FUNCTION_BLOCK "RECEIVER"	// FB 1011
TITLE = REC01
//Creation:
//Date:            Author:                                               Version
//--------------------------------------------------------------------------------
//14.04.2018     Ilia Bedniakov (ilia)                                   01.00.00
//
//Changes:
//No. Date:        Who       Description                           Mark   Version 
//--------------------------------------------------------------------------------
//01  12.01.2019  ilia       correction at comissioning            (001)  01.01.00
//
//
//_______________________________________________________________________________
//Function:
AUTHOR : ilia
NAME : project
VERSION : 0.1
VAR_INPUT
  I_iIFVacuumPumpDB : INT ;	//VacuumPump DB Nr
  I_iIFVacuumPumpDW : INT ;	//VacuumPump Interface Start DW Nr
  I_iIFStorageDB : INT ;
  I_iIFStorageDW : INT ;
  I_iIFStoLocParDB : INT ;
  I_xSystemActive : BOOL ;	//system control on
  I_xAngleValveOpen : BOOL ;	//Angle Valve Close
  I_xAngleValveClose : BOOL ;	//Angle Valve Close
  i_xPendelFlapREC : BOOL ;	//Pendulum Flap
  i_xHighLevelREC : BOOL ;	//high level sensor
  I_xPFC_PM1 : BOOL ;	//PFC PM Hopper Big Components
  I_xPFC_PM2 : BOOL ;	//PFC PM Hopper Small Components
  i_xAckFullReceiver : BOOL ;
  i_xAngleValve : BOOL ;
END_VAR
VAR_IN_OUT
  q_xAngleValve : BOOL ;	//Angle Valve Open
  q_xCleaningValve : BOOL ;	//Filter Cleaning Valve
  q_xRepperValve : BOOL ;	//Rapper Valve
  q_xRedLamp : BOOL ;
  q_xYellowLamp : BOOL ;
  q_xGreenLamp : BOOL ;
  f_xAngleValve : BOOL ;	//Angle Valve Open
  f_xFullReceiver : BOOL ;	//Fault
  f_xNoStartConditions : BOOL ;
  f_xNoPFCRequest : BOOL ;
END_VAR
VAR
  reserve_IO : ARRAY  [14 .. 49 ] OF BYTE ;
  HMI : STRUCT 	//Interface of HMI
   CMD : STRUCT
    xRelease : BOOL  := TRUE;
    xSetEmpty : BOOL ;	//VISU command button
    xAckDataSet : BOOL ;
    reserve_4 : BOOL ;
    reserve_5 : BOOL ;
    reserve_6 : BOOL ;
    reserve_7 : BOOL ;
    reserve_8 : BOOL ;
    reserve_9 : BOOL ;
    reserve_10 : BOOL ;
    reserve_11 : BOOL ;
    reserve_12 : BOOL ;
    reserve_13 : BOOL ;
    reserve : BOOL ;
    reserve_1 : BOOL ;
    reserve_2 : BOOL ;
   END_STRUCT ;
   STATE : STRUCT
    xCleaningActive : BOOL ;
    xChangeDataSetBlocked : BOOL ;
    xPFC_Request_PM1 : BOOL ;
    xPFC_Request_PM2 : BOOL ;
    xDataSetFalse : BOOL ;
    res : BOOL ;
    xFault : BOOL ;
    res_4 : BOOL ;
    res_5 : BOOL ;
    res_6 : BOOL ;
    res_7 : BOOL ;
    res_1 : BOOL ;
    res_2 : BOOL ;
    res_3 : BOOL ;
    res_8 : BOOL ;
    res_9 : BOOL ;
   END_STRUCT ;
   PARAM : STRUCT
    rCleaningDuration : REAL  := 1.500000e+001;	//cleaning pipeline dutration
    rFillingTime : REAL  := 1.000000e+001;	//Off delay for screener time
    rDischargingTime : REAL  := 3.000000e+001;	//after this time and not free LL sensor stop filling
    res_4 : REAL  := 1.000000e+001;	//Off delay for screener time
    res_4_1 : REAL  := 1.000000e+001;	//Off delay for screener time
    res_1_1 : REAL  := 3.000000e+001;	//after this time and not free LL sensor stop filling
    res_2 : REAL ;	//no new material + empty pressure -> warning
    res_3 : REAL  := 5.000000e+000;	//after enclosing HL sensor HP03 delay for discharg starts again
    iConvDataSet : INT  := 1;	//Set storage location HP01/HP02
    reserve_7 : INT ;
    reserve_8 : INT ;
    reserve_9 : INT ;
    reserve_10 : INT ;
    reserve_11 : INT ;
   END_STRUCT ;
   PV : STRUCT
    rCleaningDuration : REAL ;	//cleaning pipeline dutration
    rFillingTime : REAL ;	//Off delay for screener time
    rDischargingTime : REAL ;	//after this time and not free LL sensor stop filling
    res_2 : REAL ;	//rd for HP03
    res_2_1 : REAL ;	//rd for HP03
    res_3 : REAL ;	//Off delay for screener time
    res_4 : REAL ;	//after this time and not free LL sensor stop filling
    res_5 : REAL ;	//no new material + empty pressure -> warning
    ConvDataSet : INT ;	//Set storage location HP01/HP02
    StatusFilling : INT ;
    StatusDischarging : INT ;
    StatusREC01 : INT ;
    res_6 : INT ;
    res_7 : INT ;
   END_STRUCT ;
  END_STRUCT ;
  PROD : STRUCT 	//Interface of Production
   FROM : STRUCT
    reserve : INT ;
    reserve_1 : INT ;
    reserve_2 : INT ;
    reserve_3 : INT ;
    reserve_4 : INT ;
    reserve_5 : REAL ;
    reserve_6 : REAL ;
    CMD : STRUCT
     reserve : BOOL ;
     reserve_1 : BOOL ;
     reserve_2 : BOOL ;
     reserve_3 : BOOL ;
     reserve_4 : BOOL ;
     reserve_5 : BOOL ;
     reserve_6 : BOOL ;
     reserve_7 : BOOL ;
     reserve_8 : BOOL ;
     reserve_9 : BOOL ;
     reserve_10 : BOOL ;
     reserve_11 : BOOL ;
     reserve_12 : BOOL ;
     reserve_13 : BOOL ;
     reserve_14 : BOOL ;
     reserve_15 : BOOL ;
    END_STRUCT ;
   END_STRUCT ;
   TO : STRUCT
    reserve : INT ;
    reserve_1 : INT ;
    reserve_2 : INT ;
    reserve_3 : INT ;
    reserve_4 : INT ;
    reserve_5 : REAL ;
    reserve_6 : REAL ;
    STATE : STRUCT
     reserve : BOOL ;
     reserve_1 : BOOL ;
     reserve_2 : BOOL ;
     reserve_3 : BOOL ;
     reserve_4 : BOOL ;
     reserve_5 : BOOL ;
     reserve_6 : BOOL ;
     reserve_7 : BOOL ;
     reserve_8 : BOOL ;
     reserve_9 : BOOL ;
     reserve_10 : BOOL ;
     reserve_11 : BOOL ;
     reserve_12 : BOOL ;
     reserve_13 : BOOL ;
     reserve_14 : BOOL ;
     reserve_15 : BOOL ;
    END_STRUCT ;
   END_STRUCT ;
   reserve : ARRAY  [40 .. 49 ] OF BYTE ;
  END_STRUCT ;
  RecipeData : STRUCT
   iRecNumber : INT ;
   Recipe : STRUCT
    rSpeed : REAL ;
    rPauseTime : REAL ;
    rPulseTime : REAL ;
    reserve : ARRAY  [12 .. 49 ] OF BYTE ;
   END_STRUCT ;
  END_STRUCT ;
  reserve_HMI : ARRAY  [244 .. 299 ] OF BYTE ;
  IF_VP : STRUCT 	//Interface Blower in active object
   STATUS : STRUCT
    reserve_1 : INT ;
    reserve_2 : INT ;
    reserve_3 : INT ;
    reserve_4 : INT ;
    reserve_5 : INT ;
    rActualPressure : REAL ;
    reserve_6 : REAL ;
    STATE : STRUCT
     xReady : BOOL ;
     xActive : BOOL ;
     xPressureFault : BOOL ;
     xEmptyPressure : BOOL ;
     Fault : BOOL ;
     reserve_2 : BOOL ;
     reserve_3 : BOOL ;
     reserve_4 : BOOL ;
     reserve_5 : BOOL ;
     reserve_6 : BOOL ;
     reserve_7 : BOOL ;
     reserve_8 : BOOL ;
     reserve_9 : BOOL ;
     reserve_10 : BOOL ;
     reserve_11 : BOOL ;
     reserve_12 : BOOL ;
    END_STRUCT ;
   END_STRUCT ;
   CONTROL : STRUCT
    Answer_DB : INT ;
    Answer_DW : INT ;
    SpeedVP : INT ;
    reserve_2 : INT ;
    reserve_3 : INT ;
    reserve_4 : REAL ;
    reserve_5 : REAL ;
    CMD : STRUCT
     xRequest : BOOL ;
     xRelease : BOOL ;
     reserve : BOOL ;
     reserve_1 : BOOL ;
     reserve_2 : BOOL ;
     reserve_3 : BOOL ;
     reserve_4 : BOOL ;
     reserve_5 : BOOL ;
     reserve_6 : BOOL ;
     reserve_7 : BOOL ;
     reserve_8 : BOOL ;
     reserve_9 : BOOL ;
     reserve_10 : BOOL ;
     reserve_11 : BOOL ;
     reserve_12 : BOOL ;
     reserve_13 : BOOL ;
    END_STRUCT ;
   END_STRUCT ;
  END_STRUCT ;
  IF_Storage : STRUCT
   STATUS : STRUCT
    reserve_1 : INT ;
    reserve_2 : INT ;
    reserve_3 : INT ;
    reserve_4 : INT ;
    iRecipeNumber : INT ;
    rActualPressure : REAL ;
    reserve_6 : REAL ;
    STATE : STRUCT
     xReady : BOOL ;
     xActive : BOOL ;
     xStopped : BOOL ;
     xStarted : BOOL ;
     reserve_4 : BOOL ;
     reserve_5 : BOOL ;
     reserve_6 : BOOL ;
     reserve_7 : BOOL ;
     reserve_8 : BOOL ;
     reserve_9 : BOOL ;
     reserve_10 : BOOL ;
     reserve_11 : BOOL ;
     reserve_12 : BOOL ;
     reserve_12_1 : BOOL ;
     reserve_12_2 : BOOL ;
     reserve_12_3 : BOOL ;
    END_STRUCT ;
   END_STRUCT ;
   CONTROL : STRUCT
    Answer_DB : INT ;
    Answer_DW : INT ;
    iRecipeNumber : INT ;
    rActualPressure : REAL ;
    iPulseValve : REAL ;
    iPauseValve : REAL ;
    CMD : STRUCT
     xConnect : BOOL ;
     xRequest : BOOL ;
     xRelease : BOOL ;
     xFull : BOOL ;
     xCleaningRelease : BOOL ;
     xPressureFault : BOOL ;
     res : BOOL ;
     res_2 : BOOL ;
     xDischargeActive : BOOL ;
     res_1 : BOOL ;
     res_1_1 : BOOL ;
     res_1_2 : BOOL ;
     res_1_3 : BOOL ;
     res_1_4 : BOOL ;
     res_1_5 : BOOL ;
     res_1_6 : BOOL ;
    END_STRUCT ;
   END_STRUCT ;
  END_STRUCT ;
  reserve_IF : ARRAY  [420 .. 499 ] OF BYTE ;
  AngleValve : STRUCT 	//Angle Valve 1Q 2I
   parameter : STRUCT
    valve_on : BOOL  := TRUE;	//activate valve structure
    clock_on : BOOL ;	//activate clock structure
    reserve_3 : BOOL ;
    switching_number_on : BOOL ;	//activate switching number counter
    reserve_4 : BOOL ;
    parameter_1Q : BOOL ;	//valve type with 1 quit 0 inputs
    parameter_1Q_1I : BOOL ;	//valve type with 1 quit 1 input (=)
    parameter_1Q_1IN : BOOL ;	//valve type with 1 quit 1 input (<>)
    parameter_1Q_2I : BOOL  := TRUE;	//valve type with 1 quit 2 inputs
    parameter_text_pos_1 : BOOL ;
    parameter_text_straight : BOOL ;
    parameter_text_inverse : BOOL ;	//select text inverse = "close/open" or "bypass/convey" aso.
    parameter_text_open : BOOL ;	//select text quit = "open/close"
    parameter_text_convey : BOOL  := TRUE;	//select text quit = "convey/bypass"
    parameter_text_on : BOOL ;	//select text quit = "on/off"
    parameter_text_up : BOOL ;	//select text quit = "up/down"
   END_STRUCT ;
   quit_valve : BOOL ;	//1 = quit valve
   input_valve_set : BOOL ;	//1 = input valve, if quit valve set
   input_valve_not_set : BOOL ;	//1 = input valve, if quit valve not set
   auto_mode_control : BOOL ;	//1 = release/control of valve in auto mode
   valve_in_operation : BOOL ;	//1 = signal valve in operation
   fault : BOOL ;	//1 = signal valve fault
   man_mode_to_SCADA : BOOL ;	//0 = automatic mode , 1 = manual mode
   man_mode_from_SCADA : BOOL ;	//0 = automatic mode , 1 = manual mode
   man_mode_control : BOOL ;	//1 = release/control of valve in manual mode (from SCADA)
   man_mode_locked : BOOL ;	//1 = change to manual mode locked, valve is in automatic use
   start_with_impulse : BOOL ;	//1 = start cycle with impluse
   set_cycles_reached : BOOL ;	//1 = set number of cycles has been reached
   continous_clock : BOOL ;	//1 = continous clock / 0 = set number of clocks
   simulation : BOOL ;	//1 = simulation of object
   release_clock : BOOL ;	//1 = release bit for clock FC
   quit_clock : BOOL ;	//quit for clock FC, if release_clock = TRUE
   set_time_fault : INT  := 5;	//fault evaluation time in seconds
   actual_time_fault : INT ;	//actual fault evaluation time in seconds
   impulse_time : REAL  := 5.000000e+000;	//impulse time for clock in seconds
   break_time : REAL  := 5.000000e+000;	//break time for clock in seconds
   time_counter : REAL ;	//time counter (elapsed time)
   set_cycles : INT ;	//number of clocks if not continous clock
   clock_counter : INT ;	//clock counter
   switching_number_counter : STRUCT 	//switching number counter
    reset : BOOL ;	//reset switching number counter
    warning : BOOL ;	//warning number exceeded
    alarm : BOOL ;	//alarm number exceeded
    flank_flag : BOOL ;	//internal flag
    actual_switching_number : REAL ;	//actual switching number
    set_number_warning : REAL ;	//set number for warning
    set_number_alarm : REAL ;	//set number for alarm
   END_STRUCT ;
   set_time_in_operation : INT ;	//1IoO: set time for delay of "valve in operation"
   real_time_in_operation : INT ;	//1IoO: real time for delay of "valve in operation"
   system_on : BOOL ;	//system released resepectively system area released after emergency stopping
   reserve : ARRAY  [44 .. 47 ] OF BYTE ;
   object_state : INT ;	//1=grey; 5=green; 9=white; 15=yellow; 16=red
  END_STRUCT ;
  FilterCleaning : STRUCT 	//Angle Valve 1Q 0I
   parameter : STRUCT
    valve_on : BOOL  := TRUE;	//activate valve structure
    clock_on : BOOL ;	//activate clock structure
    reserve_3 : BOOL ;
    switching_number_on : BOOL ;	//activate switching number counter
    reserve_4 : BOOL ;
    parameter_1Q : BOOL ;	//valve type with 1 quit 0 inputs
    parameter_1Q_1I : BOOL ;	//valve type with 1 quit 1 input (=)
    parameter_1Q_1IN : BOOL ;	//valve type with 1 quit 1 input (<>)
    parameter_1Q_2I : BOOL  := TRUE;	//valve type with 1 quit 2 inputs
    parameter_text_pos_1 : BOOL ;
    parameter_text_straight : BOOL ;
    parameter_text_inverse : BOOL ;	//select text inverse = "close/open" or "bypass/convey" aso.
    parameter_text_open : BOOL ;	//select text quit = "open/close"
    parameter_text_convey : BOOL  := TRUE;	//select text quit = "convey/bypass"
    parameter_text_on : BOOL ;	//select text quit = "on/off"
    parameter_text_up : BOOL ;	//select text quit = "up/down"
   END_STRUCT ;
   quit_valve : BOOL ;	//1 = quit valve
   input_valve_set : BOOL ;	//1 = input valve, if quit valve set
   input_valve_not_set : BOOL ;	//1 = input valve, if quit valve not set
   auto_mode_control : BOOL ;	//1 = release/control of valve in auto mode
   valve_in_operation : BOOL ;	//1 = signal valve in operation
   fault : BOOL ;	//1 = signal valve fault
   man_mode_to_SCADA : BOOL ;	//0 = automatic mode , 1 = manual mode
   man_mode_from_SCADA : BOOL ;	//0 = automatic mode , 1 = manual mode
   man_mode_control : BOOL ;	//1 = release/control of valve in manual mode (from SCADA)
   man_mode_locked : BOOL ;	//1 = change to manual mode locked, valve is in automatic use
   start_with_impulse : BOOL ;	//1 = start cycle with impluse
   set_cycles_reached : BOOL ;	//1 = set number of cycles has been reached
   continous_clock : BOOL ;	//1 = continous clock / 0 = set number of clocks
   simulation : BOOL ;	//1 = simulation of object
   release_clock : BOOL ;	//1 = release bit for clock FC
   quit_clock : BOOL ;	//quit for clock FC, if release_clock = TRUE
   set_time_fault : INT  := 5;	//fault evaluation time in seconds
   actual_time_fault : INT ;	//actual fault evaluation time in seconds
   impulse_time : REAL  := 5.000000e+000;	//impulse time for clock in seconds
   break_time : REAL  := 5.000000e+000;	//break time for clock in seconds
   time_counter : REAL ;	//time counter (elapsed time)
   set_cycles : INT ;	//number of clocks if not continous clock
   clock_counter : INT ;	//clock counter
   switching_number_counter : STRUCT 	//switching number counter
    reset : BOOL ;	//reset switching number counter
    warning : BOOL ;	//warning number exceeded
    alarm : BOOL ;	//alarm number exceeded
    flank_flag : BOOL ;	//internal flag
    actual_switching_number : REAL ;	//actual switching number
    set_number_warning : REAL ;	//set number for warning
    set_number_alarm : REAL ;	//set number for alarm
   END_STRUCT ;
   set_time_in_operation : INT ;	//1IoO: set time for delay of "valve in operation"
   real_time_in_operation : INT ;	//1IoO: real time for delay of "valve in operation"
   system_on : BOOL ;	//system released resepectively system area released after emergency stopping
   reserve : ARRAY  [44 .. 47 ] OF BYTE ;
   object_state : INT ;	//1=grey; 5=green; 9=white; 15=yellow; 16=red
  END_STRUCT ;
  Rapper : STRUCT 	//Angle Valve 1Q 0I
   parameter : STRUCT
    valve_on : BOOL  := TRUE;	//activate valve structure
    clock_on : BOOL ;	//activate clock structure
    reserve_3 : BOOL ;
    switching_number_on : BOOL ;	//activate switching number counter
    reserve_4 : BOOL ;
    parameter_1Q : BOOL ;	//valve type with 1 quit 0 inputs
    parameter_1Q_1I : BOOL ;	//valve type with 1 quit 1 input (=)
    parameter_1Q_1IN : BOOL ;	//valve type with 1 quit 1 input (<>)
    parameter_1Q_2I : BOOL  := TRUE;	//valve type with 1 quit 2 inputs
    parameter_text_pos_1 : BOOL ;
    parameter_text_straight : BOOL ;
    parameter_text_inverse : BOOL ;	//select text inverse = "close/open" or "bypass/convey" aso.
    parameter_text_open : BOOL ;	//select text quit = "open/close"
    parameter_text_convey : BOOL  := TRUE;	//select text quit = "convey/bypass"
    parameter_text_on : BOOL ;	//select text quit = "on/off"
    parameter_text_up : BOOL ;	//select text quit = "up/down"
   END_STRUCT ;
   quit_valve : BOOL ;	//1 = quit valve
   input_valve_set : BOOL ;	//1 = input valve, if quit valve set
   input_valve_not_set : BOOL ;	//1 = input valve, if quit valve not set
   auto_mode_control : BOOL ;	//1 = release/control of valve in auto mode
   valve_in_operation : BOOL ;	//1 = signal valve in operation
   fault : BOOL ;	//1 = signal valve fault
   man_mode_to_SCADA : BOOL ;	//0 = automatic mode , 1 = manual mode
   man_mode_from_SCADA : BOOL ;	//0 = automatic mode , 1 = manual mode
   man_mode_control : BOOL ;	//1 = release/control of valve in manual mode (from SCADA)
   man_mode_locked : BOOL ;	//1 = change to manual mode locked, valve is in automatic use
   start_with_impulse : BOOL ;	//1 = start cycle with impluse
   set_cycles_reached : BOOL ;	//1 = set number of cycles has been reached
   continous_clock : BOOL ;	//1 = continous clock / 0 = set number of clocks
   simulation : BOOL ;	//1 = simulation of object
   release_clock : BOOL ;	//1 = release bit for clock FC
   quit_clock : BOOL ;	//quit for clock FC, if release_clock = TRUE
   set_time_fault : INT  := 5;	//fault evaluation time in seconds
   actual_time_fault : INT ;	//actual fault evaluation time in seconds
   impulse_time : REAL  := 5.000000e+000;	//impulse time for clock in seconds
   break_time : REAL  := 5.000000e+000;	//break time for clock in seconds
   time_counter : REAL ;	//time counter (elapsed time)
   set_cycles : INT ;	//number of clocks if not continous clock
   clock_counter : INT ;	//clock counter
   switching_number_counter : STRUCT 	//switching number counter
    reset : BOOL ;	//reset switching number counter
    warning : BOOL ;	//warning number exceeded
    alarm : BOOL ;	//alarm number exceeded
    flank_flag : BOOL ;	//internal flag
    actual_switching_number : REAL ;	//actual switching number
    set_number_warning : REAL ;	//set number for warning
    set_number_alarm : REAL ;	//set number for alarm
   END_STRUCT ;
   set_time_in_operation : INT ;	//1IoO: set time for delay of "valve in operation"
   real_time_in_operation : INT ;	//1IoO: real time for delay of "valve in operation"
   system_on : BOOL ;	//system released resepectively system area released after emergency stopping
   reserve : ARRAY  [44 .. 47 ] OF BYTE ;
   object_state : INT ;	//1=grey; 5=green; 9=white; 15=yellow; 16=red
  END_STRUCT ;
  BinaryObjects : STRUCT
   PendulumFlapREC01 : STRUCT
    parameter : STRUCT
     reserve : BOOL ;
     debounce_time : BOOL  := TRUE;	//view/edit debounce time
     reserve_2 : BOOL ;
     switching_number_counter : BOOL ;	//Counter for operating cycles
     reserve_4 : BOOL ;
     reserve_5 : BOOL ;
     reserve_6 : BOOL ;
     reserve_7 : BOOL ;
     parameter_invers : BOOL ;	//Parameter signal invers, invert the status
     reserve_9 : BOOL ;
     reserve_10 : BOOL ;
     reserve_11 : BOOL ;
     reserve_12 : BOOL ;
     reserve_13 : BOOL ;
     reserve_14 : BOOL ;
     reserve_15 : BOOL ;
    END_STRUCT ;
    input_processed : BOOL ;	//Input_signal processed
    input : BOOL ;	//Input signal
    def_invert_input : BOOL ;	//Definition to invert input signal (1=invert input)
    def_debounce_input : BOOL ;	//Definition to debounce input signal (1=debounce input)
    def_fault_state : BOOL ;	//Definition of fault state
    fault : BOOL ;	//1 = fault message
    man_mode_to_SCADA : BOOL ;	//0=Automode; 1=Manualmode
    man_mode_from_SCADA : BOOL ;	//0=Automode; 1=Manualmode
    man_mode_control : BOOL ;	//Control the object in manual mode (from scada)
    man_mode_locked : BOOL ;	//Lock manual mode, because object is used in auto mode
    system_on : BOOL ;
    spare : BOOL ;
    input_inverted : BOOL ;	//Input signal inverted if necessary
    input_debounced : BOOL ;	//Input signal debounced if necessary (also inverted if necessary9)
    input_debounced_high : BOOL ;	//Input signal debounced high (output signal timer)
    input_debounced_low : BOOL ;	//Input signal debounced low (output signal timer)
    set_time_fault : INT  := 5;	//Set value fault evaulation time
    act_time_fault : INT ;	//Act value fault avaulation time
    set_time_debounced_high : REAL ;
    act_time_debounced_high : REAL ;
    set_time_debounced_low : REAL ;
    act_time_debounced_low : REAL ;
    cycle_counter : STRUCT
     reset_counter : BOOL ;	//Reset operating cycle counter
     warning : BOOL ;	//Warning time 1 elapsed
     alarm : BOOL ;	//Alarm time 2 elapsed
     flank_flag : BOOL ;	//Intern used flag
     act_number_of_cycles : REAL ;	//Actual number of cycles (cycle counter)
     set_number_warning : REAL ;	//Set value for generate the warning
     set_number_alarm : REAL ;	//Set value for generate the alarm
    END_STRUCT ;
    reserve : ARRAY  [38 .. 47 ] OF BYTE ;
    object_state : INT ;
   END_STRUCT ;
   HighLevelREC01 : STRUCT
    parameter : STRUCT
     reserve : BOOL ;
     debounce_time : BOOL  := TRUE;	//view/edit debounce time
     reserve_2 : BOOL ;
     switching_number_counter : BOOL ;	//Counter for operating cycles
     reserve_4 : BOOL ;
     reserve_5 : BOOL ;
     reserve_6 : BOOL ;
     reserve_7 : BOOL ;
     parameter_invers : BOOL ;	//Parameter signal invers, invert the status
     reserve_9 : BOOL ;
     reserve_10 : BOOL ;
     reserve_11 : BOOL ;
     reserve_12 : BOOL ;
     reserve_13 : BOOL ;
     reserve_14 : BOOL ;
     reserve_15 : BOOL ;
    END_STRUCT ;
    input_processed : BOOL ;	//Input_signal processed
    input : BOOL ;	//Input signal
    def_invert_input : BOOL ;	//Definition to invert input signal (1=invert input)
    def_debounce_input : BOOL ;	//Definition to debounce input signal (1=debounce input)
    def_fault_state : BOOL ;	//Definition of fault state
    fault : BOOL ;	//1 = fault message
    man_mode_to_SCADA : BOOL ;	//0=Automode; 1=Manualmode
    man_mode_from_SCADA : BOOL ;	//0=Automode; 1=Manualmode
    man_mode_control : BOOL ;	//Control the object in manual mode (from scada)
    man_mode_locked : BOOL ;	//Lock manual mode, because object is used in auto mode
    system_on : BOOL ;
    spare : BOOL ;
    input_inverted : BOOL ;	//Input signal inverted if necessary
    input_debounced : BOOL ;	//Input signal debounced if necessary (also inverted if necessary9)
    input_debounced_high : BOOL ;	//Input signal debounced high (output signal timer)
    input_debounced_low : BOOL ;	//Input signal debounced low (output signal timer)
    set_time_fault : INT  := 5;	//Set value fault evaulation time
    act_time_fault : INT ;	//Act value fault avaulation time
    set_time_debounced_high : REAL ;
    act_time_debounced_high : REAL ;
    set_time_debounced_low : REAL ;
    act_time_debounced_low : REAL ;
    cycle_counter : STRUCT
     reset_counter : BOOL ;	//Reset operating cycle counter
     warning : BOOL ;	//Warning time 1 elapsed
     alarm : BOOL ;	//Alarm time 2 elapsed
     flank_flag : BOOL ;	//Intern used flag
     act_number_of_cycles : REAL ;	//Actual number of cycles (cycle counter)
     set_number_warning : REAL ;	//Set value for generate the warning
     set_number_alarm : REAL ;	//Set value for generate the alarm
    END_STRUCT ;
    reserve : ARRAY  [38 .. 47 ] OF BYTE ;
    object_state : INT ;
   END_STRUCT ;
   PFC_PM1 : STRUCT
    parameter : STRUCT
     reserve : BOOL ;
     debounce_time : BOOL  := TRUE;	//view/edit debounce time
     reserve_2 : BOOL ;
     switching_number_counter : BOOL ;	//Counter for operating cycles
     reserve_4 : BOOL ;
     reserve_5 : BOOL ;
     reserve_6 : BOOL ;
     reserve_7 : BOOL ;
     parameter_invers : BOOL ;	//Parameter signal invers, invert the status
     reserve_9 : BOOL ;
     reserve_10 : BOOL ;
     reserve_11 : BOOL ;
     reserve_12 : BOOL ;
     reserve_13 : BOOL ;
     reserve_14 : BOOL ;
     reserve_15 : BOOL ;
    END_STRUCT ;
    input_processed : BOOL ;	//Input_signal processed
    input : BOOL ;	//Input signal
    def_invert_input : BOOL ;	//Definition to invert input signal (1=invert input)
    def_debounce_input : BOOL ;	//Definition to debounce input signal (1=debounce input)
    def_fault_state : BOOL ;	//Definition of fault state
    fault : BOOL ;	//1 = fault message
    man_mode_to_SCADA : BOOL ;	//0=Automode; 1=Manualmode
    man_mode_from_SCADA : BOOL ;	//0=Automode; 1=Manualmode
    man_mode_control : BOOL ;	//Control the object in manual mode (from scada)
    man_mode_locked : BOOL ;	//Lock manual mode, because object is used in auto mode
    system_on : BOOL ;
    spare : BOOL ;
    input_inverted : BOOL ;	//Input signal inverted if necessary
    input_debounced : BOOL ;	//Input signal debounced if necessary (also inverted if necessary9)
    input_debounced_high : BOOL ;	//Input signal debounced high (output signal timer)
    input_debounced_low : BOOL ;	//Input signal debounced low (output signal timer)
    set_time_fault : INT  := 5;	//Set value fault evaulation time
    act_time_fault : INT ;	//Act value fault avaulation time
    set_time_debounced_high : REAL ;
    act_time_debounced_high : REAL ;
    set_time_debounced_low : REAL ;
    act_time_debounced_low : REAL ;
    cycle_counter : STRUCT
     reset_counter : BOOL ;	//Reset operating cycle counter
     warning : BOOL ;	//Warning time 1 elapsed
     alarm : BOOL ;	//Alarm time 2 elapsed
     flank_flag : BOOL ;	//Intern used flag
     act_number_of_cycles : REAL ;	//Actual number of cycles (cycle counter)
     set_number_warning : REAL ;	//Set value for generate the warning
     set_number_alarm : REAL ;	//Set value for generate the alarm
    END_STRUCT ;
    reserve : ARRAY  [38 .. 47 ] OF BYTE ;
    object_state : INT ;
   END_STRUCT ;
   PFC_PM2 : STRUCT
    parameter : STRUCT
     reserve : BOOL ;
     debounce_time : BOOL  := TRUE;	//view/edit debounce time
     reserve_2 : BOOL ;
     switching_number_counter : BOOL ;	//Counter for operating cycles
     reserve_4 : BOOL ;
     reserve_5 : BOOL ;
     reserve_6 : BOOL ;
     reserve_7 : BOOL ;
     parameter_invers : BOOL ;	//Parameter signal invers, invert the status
     reserve_9 : BOOL ;
     reserve_10 : BOOL ;
     reserve_11 : BOOL ;
     reserve_12 : BOOL ;
     reserve_13 : BOOL ;
     reserve_14 : BOOL ;
     reserve_15 : BOOL ;
    END_STRUCT ;
    input_processed : BOOL ;	//Input_signal processed
    input : BOOL ;	//Input signal
    def_invert_input : BOOL ;	//Definition to invert input signal (1=invert input)
    def_debounce_input : BOOL ;	//Definition to debounce input signal (1=debounce input)
    def_fault_state : BOOL ;	//Definition of fault state
    fault : BOOL ;	//1 = fault message
    man_mode_to_SCADA : BOOL ;	//0=Automode; 1=Manualmode
    man_mode_from_SCADA : BOOL ;	//0=Automode; 1=Manualmode
    man_mode_control : BOOL ;	//Control the object in manual mode (from scada)
    man_mode_locked : BOOL ;	//Lock manual mode, because object is used in auto mode
    system_on : BOOL ;
    spare : BOOL ;
    input_inverted : BOOL ;	//Input signal inverted if necessary
    input_debounced : BOOL ;	//Input signal debounced if necessary (also inverted if necessary9)
    input_debounced_high : BOOL ;	//Input signal debounced high (output signal timer)
    input_debounced_low : BOOL ;	//Input signal debounced low (output signal timer)
    set_time_fault : INT  := 5;	//Set value fault evaulation time
    act_time_fault : INT ;	//Act value fault avaulation time
    set_time_debounced_high : REAL ;
    act_time_debounced_high : REAL ;
    set_time_debounced_low : REAL ;
    act_time_debounced_low : REAL ;
    cycle_counter : STRUCT
     reset_counter : BOOL ;	//Reset operating cycle counter
     warning : BOOL ;	//Warning time 1 elapsed
     alarm : BOOL ;	//Alarm time 2 elapsed
     flank_flag : BOOL ;	//Intern used flag
     act_number_of_cycles : REAL ;	//Actual number of cycles (cycle counter)
     set_number_warning : REAL ;	//Set value for generate the warning
     set_number_alarm : REAL ;	//Set value for generate the alarm
    END_STRUCT ;
    reserve : ARRAY  [38 .. 47 ] OF BYTE ;
    object_state : INT ;
   END_STRUCT ;
  END_STRUCT ;
  reserve_Cmod : ARRAY  [850 .. 949 ] OF BYTE ;
  TIMERS : STRUCT 	//ten timers
   TON_Cleaning : STRUCT
    IN : BOOL ;
    RST : BOOL ;
    IMP : BOOL ;
    Q : BOOL ;
    PT : REAL ;
    ET : REAL ;
   END_STRUCT ;
   TON_FillingTime : STRUCT
    IN : BOOL ;
    RST : BOOL ;
    IMP : BOOL ;
    Q : BOOL ;
    PT : REAL ;
    ET : REAL ;
   END_STRUCT ;
   TON_DischargingTime : STRUCT
    IN : BOOL ;
    RST : BOOL ;
    IMP : BOOL ;
    Q : BOOL ;
    PT : REAL ;
    ET : REAL ;
   END_STRUCT ;
   res_Timer_1 : STRUCT
    IN : BOOL ;
    RST : BOOL ;
    IMP : BOOL ;
    Q : BOOL ;
    PT : REAL ;
    ET : REAL ;
   END_STRUCT ;
   res_Timer_2 : STRUCT
    IN : BOOL ;
    RST : BOOL ;
    IMP : BOOL ;
    Q : BOOL ;
    PT : REAL ;
    ET : REAL ;
   END_STRUCT ;
   res_Timer_2_1 : STRUCT
    IN : BOOL ;
    RST : BOOL ;
    IMP : BOOL ;
    Q : BOOL ;
    PT : REAL ;
    ET : REAL ;
   END_STRUCT ;
  END_STRUCT ;
  SEQUENCES : STRUCT
   Filling : STRUCT
    AUTO : BOOL ;
    MANUAL : BOOL ;
    LOCKED : BOOL ;
    RELEASE : BOOL ;
    ACTIVE : BOOL ;
    CLEANING : BOOL ;
    FAULTED : BOOL ;
    reserve_4 : BOOL ;
    reserve_5 : BOOL ;
    reserve_6 : BOOL ;
    reserve_7 : BOOL ;
    reserve_8 : BOOL ;
    reserve_9 : BOOL ;
    reserve_10 : BOOL ;
    reserve_11 : BOOL ;
    reserve_12 : BOOL ;
   END_STRUCT ;
   Discharging : STRUCT
    AUTO : BOOL ;
    MANUAL : BOOL ;
    LOCKED : BOOL ;
    RELEASE : BOOL ;
    ACTIVE : BOOL ;
    RESTDISCHARGE_REQ : BOOL ;
    reserve_1 : BOOL ;
    FAULTED : BOOL ;
    reserve_5 : BOOL ;
    reserve_6 : BOOL ;
    reserve_7 : BOOL ;
    reserve_8 : BOOL ;
    reserve_9 : BOOL ;
    reserve_10 : BOOL ;
    reserve_11 : BOOL ;
    reserve_12 : BOOL ;
   END_STRUCT ;
   reserve : ARRAY  [4 .. 99 ] OF BYTE ;
  END_STRUCT ;
  INTERNAL : STRUCT
   IF : STRUCT
    Storage : STRUCT
     StorageLocationNumber : INT ;
     StorageLocation_DB : INT ;
     StorageLocation_DW : INT ;
     reserve : INT ;
     res : BOOL ;
     IF_Silo_free : BOOL ;
     res_1 : BOOL ;
     res_2 : BOOL ;
     res_3 : BOOL ;
     res_4 : BOOL ;
     res_5 : BOOL ;
     res_6 : BOOL ;
    END_STRUCT ;
    Blower : STRUCT
     Blower_DB : INT ;
     Blower_DW : INT ;
     reserve : INT ;
     Blower_ready : BOOL ;
     Blower_free : BOOL ;
     reserve_2 : BOOL ;
     reserve_3 : BOOL ;
     reserve_1_1 : BOOL ;
     reserve_2_1 : BOOL ;
     reserve_3_1 : BOOL ;
     reserve_3_1_1 : BOOL ;
    END_STRUCT ;
    FC_RF : STRUCT
     RF_DB : INT ;
     RF_DW : INT ;
     reserve : INT ;
     RF_ready : BOOL ;
     RF_free : BOOL ;
     res : BOOL ;
     res_1 : BOOL ;
     res_2 : BOOL ;
     res_3 : BOOL ;
     res_4 : BOOL ;
     res_5 : BOOL ;
    END_STRUCT ;
    reserve_6 : BOOL ;
    reserve_7 : BOOL ;
    reserve_8 : BOOL ;
    reserve_9 : BOOL ;
    reserve_10 : BOOL ;
    reserve_11 : BOOL ;
    reserve_12 : BOOL ;
   END_STRUCT ;
   Flags : STRUCT
    FP_FalseDataset : STRUCT
     helpBit : BOOL ;
     pulseBit : BOOL ;
    END_STRUCT ;
    FP_CleaningRelease : STRUCT
     helpBit : BOOL ;
     pulseBit : BOOL ;
    END_STRUCT ;
    StatusREC : STRUCT
     xFilled : BOOL ;
     xFull : BOOL ;
     xEmpty : BOOL ;
     res : BOOL ;
     res_1 : BOOL ;
     res_2 : BOOL ;
     res_3 : BOOL ;
     res_4 : BOOL ;
    END_STRUCT ;
    BUTTONS_LAMPS : STRUCT
     LMStart : STRUCT
      Steady : BOOL ;
      Flash : BOOL ;
      DoubleFlash : BOOL ;
      Activated : BOOL ;
      res_1 : BOOL ;
      res_2 : BOOL ;
      res_3 : BOOL ;
      res_4 : BOOL ;
     END_STRUCT ;
     LMStop : STRUCT
      Steady : BOOL ;
      Flash : BOOL ;
      DoubleFlash : BOOL ;
      Activated : BOOL ;
      res_1 : BOOL ;
      res_2 : BOOL ;
      res_3 : BOOL ;
      res_4 : BOOL ;
     END_STRUCT ;
     Green : STRUCT
      Steady : BOOL ;
      Flash : BOOL ;
      DoubleFlash : BOOL ;
      res : BOOL ;
      res_1 : BOOL ;
      res_2 : BOOL ;
      res_3 : BOOL ;
      res_4 : BOOL ;
     END_STRUCT ;
     Yellow : STRUCT
      Steady : BOOL ;
      Flash : BOOL ;
      DoubleFlash : BOOL ;
      res : BOOL ;
      res_1 : BOOL ;
      res_2 : BOOL ;
      res_3 : BOOL ;
      res_4 : BOOL ;
     END_STRUCT ;
     Red : STRUCT
      Steady : BOOL ;
      Flash : BOOL ;
      DoubleFlash : BOOL ;
      res : BOOL ;
      res_1 : BOOL ;
      res_2 : BOOL ;
      res_3 : BOOL ;
      res_4 : BOOL ;
     END_STRUCT ;
     res_5 : BOOL ;
     res_1_1 : BOOL ;
     res_2_1 : BOOL ;
     res_3_1 : BOOL ;
     res_4_1 : BOOL ;
     res : BOOL ;
     res_1 : BOOL ;
     res_2 : BOOL ;
    END_STRUCT ;
    Switches : STRUCT
     xPendulumFlapClosed : BOOL ;
     xHighLevelCovered : BOOL ;
     ress : BOOL ;
     res_2 : BOOL ;
     res_3 : BOOL ;
     res_4 : BOOL ;
     res_5 : BOOL ;
     res_6 : BOOL ;
    END_STRUCT ;
    xStoLocParTaken : BOOL ;
    xPipeCleaned : BOOL ;
    xStartNewDatSet : BOOL ;
    xRequestPM : BOOL ;
    res_1 : BOOL ;
    res_2 : BOOL ;
    res_3 : BOOL ;
    res_4 : BOOL ;
    iCurrentRecipeNumber : INT ;
    iRes : BOOL ;
   END_STRUCT ;
   Instance_DB_number : INT ;
   ConveyingDataSet : STRUCT
    RecipeNumber : INT ;
    RecipeData : STRUCT 	//Recipe 1
     RecipeName : STRING  [18 ];	//Recipe Name
     SpeedRinne : INT ;	//Speed of Rinne
     reserve : INT ;	//Speed of RF
     SpeedVacuumPump : INT ;	//Speed of VP1
     NumberPumps : INT ;
     reserve1 : INT ;
     reserve2 : INT ;
     reserve3 : ARRAY  [1 .. 6 ] OF BYTE  := B#16#0;
    END_STRUCT ;
   END_STRUCT ;
  END_STRUCT ;
END_VAR
VAR_TEMP
  StorageLoc_List_DW : INT ;
  StorageLocCopyError : INT ;
  tempDB : INT ;
  OffsetAddresse : INT ;
  outFault : INT ;
  dummyBOOL : BOOL ;
  silonumbertest : STRUCT
   silo1 : INT ;
   silo2 : INT ;
  END_STRUCT ;
END_VAR
BEGIN
NETWORK
TITLE = ------------------ INSTANCE DB (STANDART)-----------------------
      L     0;
      L     DINO;
      ==I;
      BEC;
      T     #INTERNAL.Instance_DB_number;
NETWORK
TITLE = ----------------SEQUENCES AUTO/LOCKED/MANUAL-----------------
NETWORK
TITLE = Sequence discharging auto
      AN    #SEQUENCES.Discharging.LOCKED;
      =     #SEQUENCES.Discharging.AUTO;
NETWORK
TITLE = Sequence discharging manual
//should be (ilia)
      CLR;
      =     #SEQUENCES.Discharging.MANUAL;
NETWORK
TITLE = Sequence discharging locked
      O     #SEQUENCES.Discharging.MANUAL;
      ON    #I_xSystemActive;
      =     #SEQUENCES.Discharging.LOCKED;
NETWORK
TITLE = Sequence filling auto
      AN    #SEQUENCES.Filling.LOCKED;
      =     #SEQUENCES.Filling.AUTO;
NETWORK
TITLE = Sequence filling manual
//manual = important motor is in manual, e.g. Rotary valve, screw, but in other 
//case CLR. Here angle valve is main part of unit
//AN    #SEQUENCES.Filling.AUTO
      O     #AngleValve.man_mode_to_SCADA;
      =     #SEQUENCES.Filling.MANUAL;
NETWORK
TITLE = Sequence filling locked
      AN    #I_xSystemActive;
      O     #SEQUENCES.Filling.MANUAL;
      =     #SEQUENCES.Filling.LOCKED;
NETWORK
TITLE = ---------------------SENSORS/SWITCHES --------------------------
NETWORK
TITLE = Pendulum Flap REC01
      CALL  "FC24 Binär-E" (
           in_Handbedienung_erlaubt := TRUE,
           in_Anlage_ein            := #I_xSystemActive,
           in_Eingang               := #i_xPendelFlapREC,
           in_Eingang_drehen        := FALSE,
           in_Eingang_entprellen    := TRUE,
           in_Stoerauswertung_aktiv := FALSE,
           in_Quitt_Stoerung_noetig := FALSE,
           in_Stoer_Zustand         := FALSE,
           in_Quitt_Stoerung        := FALSE,
           io_Eingang_verarbeitet   := #INTERNAL.Flags.Switches.xPendulumFlapClosed,
           io_Stoerung              := #BinaryObjects.PendulumFlapREC01.fault,
           io_Struktur              := #BinaryObjects.PendulumFlapREC01);	// close is close / no needed faultys
NETWORK
TITLE = High Level Sensor REC01
      CALL  "FC24 Binär-E" (
           in_Handbedienung_erlaubt := TRUE,
           in_Anlage_ein            := #I_xSystemActive,
           in_Eingang               := #i_xHighLevelREC,
           in_Eingang_drehen        := TRUE,
           in_Eingang_entprellen    := TRUE,
           in_Stoerauswertung_aktiv := TRUE,
           in_Quitt_Stoerung_noetig := FALSE,
           in_Stoer_Zustand         := FALSE,
           in_Quitt_Stoerung        := FALSE,
           io_Eingang_verarbeitet   := #INTERNAL.Flags.Switches.xHighLevelCovered,
           io_Stoerung              := #f_xFullReceiver,
           io_Struktur              := #BinaryObjects.HighLevelREC01);
NETWORK
TITLE = -----------------------INPUT  PFC ------------------------------
NETWORK
TITLE = Discharging: Internal Request from PM
      O     #I_xPFC_PM1;
      O     #I_xPFC_PM2;
      =     #INTERNAL.Flags.xRequestPM;
NETWORK
TITLE = ----------------START NEW RECIPE------------------------------
NETWORK
TITLE = False Recipe number (Conveying Parameters)
//recipe =0
//OR
//new recipe AND REC NOT empty
//OR
//recipeREC <> REC CST
      A(;
      L     #HMI.PARAM.iConvDataSet;
      L     0;
      ==I;
      );
      O;
      A(;
      L     #HMI.PARAM.iConvDataSet;
      L     #IF_Storage.STATUS.iRecipeNumber;
      <>I;
      );
      AN    #INTERNAL.Flags.StatusREC.xEmpty;
      O;
      A(;
      L     #HMI.PARAM.iConvDataSet;
      L     #IF_Storage.STATUS.iRecipeNumber;
      <>I;
      );
      S     #HMI.STATE.xDataSetFalse;
      A     #HMI.CMD.xAckDataSet;
      R     #HMI.STATE.xDataSetFalse;
NETWORK
TITLE = Start new recipe
      AN    #HMI.STATE.xDataSetFalse;
      A     #INTERNAL.Flags.StatusREC.xEmpty;
      O;
      A(;
      L     #INTERNAL.Flags.iCurrentRecipeNumber;
      L     #IF_Storage.STATUS.iRecipeNumber;
      ==I;
      );
      S     #INTERNAL.Flags.xStartNewDatSet;
      AN    #SEQUENCES.Filling.ACTIVE;
      AN    #SEQUENCES.Filling.CLEANING;
      A     #INTERNAL.Flags.StatusREC.xEmpty;
      O     #HMI.STATE.xDataSetFalse;
      R     #INTERNAL.Flags.xStartNewDatSet;
//TODO TO LOOK
      R     #INTERNAL.Flags.xStoLocParTaken;
NETWORK
TITLE = Actual Recipe REC01
//New Data set - > Current Recipe
      A     #INTERNAL.Flags.xStartNewDatSet;
      FP    #INTERNAL.Flags.FP_FalseDataset.helpBit;
      L     #HMI.PARAM.iConvDataSet;
      JCN   WRA;	//write Recipe
      T     #INTERNAL.Flags.iCurrentRecipeNumber;
WRA:  NOP   0;
NETWORK
TITLE = Wrong start sequence - FAULT
      ON    #I_xSystemActive;
      O     #HMI.STATE.xDataSetFalse;
      O;
      A     #INTERNAL.Flags.xStartNewDatSet;
      A     #IF_Storage.CONTROL.CMD.xRequest;
      AN    #IF_Storage.STATUS.STATE.xReady;
      O;
      AN    #INTERNAL.Flags.StatusREC.xEmpty;
      =     #f_xNoStartConditions;
NETWORK
TITLE = Block HMI Button for new Recipe 
      O     #SEQUENCES.Filling.ACTIVE;
      O     #SEQUENCES.Discharging.ACTIVE;
      =     #HMI.STATE.xChangeDataSetBlocked;
NETWORK
TITLE = Take Storage Location
//MUST BE TAKEN FROM RECIPE DB
      A     #INTERNAL.Flags.xStartNewDatSet;
      AN    #INTERNAL.Flags.xStoLocParTaken;
      JCN   SLT;	// storage location take
      L     #HMI.PARAM.iConvDataSet;
      L     1;
      -I;
      L     40;
      *I;
      T     #INTERNAL.IF.Storage.StorageLocation_DW;
      L     1;
      T     #INTERNAL.IF.Storage.StorageLocationNumber;
      L     #I_iIFStoLocParDB;
      T     #INTERNAL.IF.Storage.StorageLocation_DB;
      CALL  "FC7 Tabelle auslesen" (
           in_Tabelle_DB            := #INTERNAL.IF.Storage.StorageLocation_DB,
           in_Offset_DW             := #INTERNAL.IF.Storage.StorageLocation_DW,
           in_Zeile_lesen           := #INTERNAL.IF.Storage.StorageLocationNumber,
           out_Fehler               := #outFault,
           io_Ziel                  := #INTERNAL.ConveyingDataSet.RecipeData);
      A     #INTERNAL.Flags.xStartNewDatSet;
      =     #INTERNAL.Flags.xStoLocParTaken;
      L     #HMI.PARAM.iConvDataSet;
      T     #HMI.PV.ConvDataSet;
SLT:  NOP   0;
NETWORK
TITLE = -------------SEQUENCES/HANDSHAKES FILLING --------------------
NETWORK
TITLE = Filling: Request to CST01
      A     #SEQUENCES.Filling.AUTO;
      A     #HMI.CMD.xRelease;
      A     #INTERNAL.Flags.xStartNewDatSet;
      =     #IF_Storage.CONTROL.CMD.xRequest;
NETWORK
TITLE = Filling: RELEASE SEQ
//Ready from Storage - BtnStart
//Request to Storage - HMI Release
      A     #SEQUENCES.Filling.AUTO;
      A     #IF_Storage.CONTROL.CMD.xRequest;
      A     #IF_Storage.STATUS.STATE.xReady;
      AN    #SEQUENCES.Discharging.RELEASE;
      AN    #SEQUENCES.Filling.CLEANING;
      AN    #INTERNAL.Flags.Switches.xHighLevelCovered;
      S     #SEQUENCES.Filling.RELEASE;
      A     #SEQUENCES.Discharging.RELEASE;
      O     #INTERNAL.Flags.StatusREC.xEmpty;
      O     #TIMERS.TON_FillingTime.Q;
//    O     #IF_Storage.STATUS.STATE.xStopped
      ON    #IF_Storage.STATUS.STATE.xReady;
      R     #SEQUENCES.Filling.RELEASE;
NETWORK
TITLE = Filling: Filling Time
      A     #SEQUENCES.Filling.RELEASE;
      =     #TIMERS.TON_FillingTime.IN;
      CALL  "FC3 Timernachbildung" (
           in_Freigabe              := #TIMERS.TON_FillingTime.IN,
           in_Reset                 := #TIMERS.TON_FillingTime.RST,
           in_Impuls                := "M1.7 ClockTimerFunction",
           in_Impulszeit_in_100ms   := "MW 6 Timer Val Cycle FCs",
           in_Verzoegerungsart      := B#16#45,
           in_Verzoegerungszeit     := #HMI.PARAM.rFillingTime,
           io_Ausgangssignal        := #TIMERS.TON_FillingTime.Q,
           io_Zeitzaehler           := #TIMERS.TON_DischargingTime.ET);
NETWORK
TITLE = Filling: CLEANING SEQ (Pipe cleaned BIT)
//Cleaned Reset
      A     #IF_Storage.STATUS.STATE.xActive;
      R     #INTERNAL.Flags.xPipeCleaned;
      A     #IF_Storage.STATUS.STATE.xStopped;
      AN    #INTERNAL.Flags.xPipeCleaned;
      O;
      A     #SEQUENCES.Filling.CLEANING;
      AN    #INTERNAL.Flags.xPipeCleaned;
      AN    #IF_Storage.CONTROL.CMD.xRelease;
      =     #SEQUENCES.Filling.CLEANING;
// Timer for sequence
      A     #SEQUENCES.Filling.CLEANING;
      =     #TIMERS.TON_Cleaning.IN;
      ON    #I_xSystemActive;
      =     #TIMERS.TON_Cleaning.RST;
      CALL  "FC3 Timernachbildung" (
           in_Freigabe              := #TIMERS.TON_Cleaning.IN,
           in_Reset                 := #TIMERS.TON_Cleaning.RST,
           in_Impuls                := "M1.7 ClockTimerFunction",
           in_Impulszeit_in_100ms   := "MW 6 Timer Val Cycle FCs",
           in_Verzoegerungsart      := B#16#45,
           in_Verzoegerungszeit     := #HMI.PARAM.rCleaningDuration,
           io_Ausgangssignal        := #TIMERS.TON_Cleaning.Q,
           io_Zeitzaehler           := #TIMERS.TON_Cleaning.ET);
// right time to the HMI
      A     #TIMERS.TON_Cleaning.IN;
      AN    #TIMERS.TON_Cleaning.Q;
      L     0.000000e+00;
      JCN   RTH2;	//right time to HMI 
      L     #TIMERS.TON_Cleaning.ET;
RTH2: T     #HMI.PV.rCleaningDuration;
// set help Bit
      A     #TIMERS.TON_Cleaning.Q;
      S     #INTERNAL.Flags.xPipeCleaned;
NETWORK
TITLE = Filling: Request BLOWER IF
      O     #SEQUENCES.Filling.RELEASE;
      O     #SEQUENCES.Filling.CLEANING;
      =     #IF_VP.CONTROL.CMD.xRequest;
NETWORK
TITLE = Filling: Frequency to BLOWER IF
      A     #IF_VP.CONTROL.CMD.xRequest;
      A     #IF_VP.STATUS.STATE.xReady;
      JCN   NBR;	// no request
      L     #INTERNAL.ConveyingDataSet.RecipeData.SpeedVacuumPump;
      T     #IF_VP.CONTROL.SpeedVP;
NBR:  NOP   0;
NETWORK
TITLE = Filling: Release BLOWER IF 
      A(;
      O     #SEQUENCES.Filling.RELEASE;
      O     #SEQUENCES.Filling.CLEANING;
      );
      A     #IF_VP.CONTROL.CMD.xRequest;
      A     #IF_VP.STATUS.STATE.xReady;
      =     #IF_VP.CONTROL.CMD.xRelease;
NETWORK
TITLE = Filling: Release STORAGE IF
//the condition about HP full has to be checked - may be it is necessary
      A     #SEQUENCES.Filling.RELEASE;
      AN    #INTERNAL.Flags.StatusREC.xFull;
      A     #IF_Storage.STATUS.STATE.xReady;
      A     #IF_VP.STATUS.STATE.xActive;
      AN    #IF_VP.STATUS.STATE.xPressureFault;
      A     #INTERNAL.Flags.xStoLocParTaken;
      AN    #IF_VP.STATUS.STATE.xPressureFault;
      =     #IF_Storage.CONTROL.CMD.xRelease;
NETWORK
TITLE = Filling: Actual Pressure to Storage
      L     #IF_VP.STATUS.rActualPressure;
      T     #IF_Storage.CONTROL.rActualPressure;
NETWORK
TITLE = Filling: Cleaning/Pressure/SF Full  to STORAGE IF
      A     #SEQUENCES.Filling.CLEANING;
      =     #IF_Storage.CONTROL.CMD.xCleaningRelease;
NETWORK
TITLE = Filling: FAULTED to STORAGE IF
//O     #fHP01HighLevel
      O     #IF_VP.STATUS.STATE.xPressureFault;
      O     #IF_VP.STATUS.STATE.Fault;
      =     #SEQUENCES.Filling.FAULTED;
NETWORK
TITLE = Filling: FILLING ACTIVE SEQ
      A(;
      O     #SEQUENCES.Filling.RELEASE;
      O     #SEQUENCES.Filling.CLEANING;
      );
      A     #IF_VP.STATUS.STATE.xActive;
      A     #IF_Storage.STATUS.STATE.xActive;
      =     #SEQUENCES.Filling.ACTIVE;
NETWORK
TITLE = -------------SEQUENCES/HANDSHAKES DISCHARGING ------------
NETWORK
TITLE = Discharging: Discharging SEQ RELEASE (with timer)
      A     #SEQUENCES.Discharging.AUTO;
      A     #I_xSystemActive;
      A     #INTERNAL.Flags.StatusREC.xFilled;
      AN    #SEQUENCES.Filling.RELEASE;
      AN    #SEQUENCES.Filling.CLEANING;
      O;
      A     #INTERNAL.Flags.Switches.xHighLevelCovered;
      =     #SEQUENCES.Filling.RELEASE;
      A     #SEQUENCES.Filling.RELEASE;
      =     #TIMERS.TON_DischargingTime.IN;
      CALL  "FC3 Timernachbildung" (
           in_Freigabe              := #TIMERS.TON_DischargingTime.IN,
           in_Reset                 := #TIMERS.TON_DischargingTime.RST,
           in_Impuls                := "M1.7 ClockTimerFunction",
           in_Impulszeit_in_100ms   := "MW 6 Timer Val Cycle FCs",
           in_Verzoegerungsart      := B#16#45,
           in_Verzoegerungszeit     := #HMI.PARAM.rDischargingTime,
           io_Ausgangssignal        := #TIMERS.TON_DischargingTime.Q,
           io_Zeitzaehler           := #TIMERS.TON_DischargingTime.ET);
// Timer to HMI
NETWORK
TITLE = Discharging: DISCHARGING ACTIVE
      A     #SEQUENCES.Discharging.AUTO;
      A(;
      O     #SEQUENCES.Discharging.RELEASE;
      O     #SEQUENCES.Discharging.RESTDISCHARGE_REQ;
      );
      =     #SEQUENCES.Discharging.ACTIVE;
      A     #SEQUENCES.Discharging.ACTIVE;
      =     #IF_Storage.CONTROL.CMD.xDischargeActive;
NETWORK
TITLE = -------------AGGREGATES ------------
NETWORK
TITLE = Filling: Angle Valve
      A     #SEQUENCES.Filling.RELEASE;
      O     #SEQUENCES.Filling.CLEANING;
      =     #AngleValve.auto_mode_control;
      A     #AngleValve.auto_mode_control;
//      AN    "Service Mode ExpertMode"
      =     #AngleValve.man_mode_locked;
      CALL  "FC21 Ventil 1A0-2E" (
           in_Ventil_Typ            := 1,
           in_Handbedienung_erlaubt := "Release Man Mode Valves",
           in_Quitt_Stoerung_noetig := "AckObligatoryValves",
           in_Quitt_Stoerung        := #i_xAngleValve,
           in_Anlage_ein            := #I_xSystemActive,
           in_Ansteuerung_Ventil    := #AngleValve.auto_mode_control,
           in_Eingang_angesteuert   := #I_xAngleValveOpen,
           in_Eingang_nicht_angest  := #I_xAngleValveClose,
           io_Ausgang_Ventil        := #q_xAngleValve,
           io_Ventil_in_Betrieb     := #AngleValve.valve_in_operation,
           io_Stoerung              := #AngleValve.fault,
           io_Ventilstruktur        := #AngleValve);
NETWORK
TITLE = Filling/Discharging: FilterCleaning Valve
      A     #SEQUENCES.Filling.RELEASE;
      O     #SEQUENCES.Filling.CLEANING;
      =     #FilterCleaning.auto_mode_control;
// man mode locked
      A     #FilterCleaning.auto_mode_control;
      AN    "Service Mode ExpertMode";
      =     #FilterCleaning.man_mode_locked;
      CALL  "FC21 Ventil 1A0-2E" (
           in_Ventil_Typ            := 0,
           in_Handbedienung_erlaubt := TRUE,
           in_Quitt_Stoerung_noetig := FALSE,
           in_Quitt_Stoerung        := TRUE,
           in_Anlage_ein            := #I_xSystemActive,
           in_Ansteuerung_Ventil    := #FilterCleaning.auto_mode_control,
           in_Eingang_angesteuert   := FALSE,
           in_Eingang_nicht_angest  := FALSE,
           io_Ausgang_Ventil        := #q_xCleaningValve,
           io_Ventil_in_Betrieb     := #FilterCleaning.valve_in_operation,
           io_Stoerung              := #FilterCleaning.fault,
           io_Ventilstruktur        := #FilterCleaning);
NETWORK
TITLE = Discharging: RapperValve
      A     #SEQUENCES.Discharging.RELEASE;
      =     #Rapper.auto_mode_control;
// man mode locked
      A     #Rapper.auto_mode_control;
      AN    "Service Mode ExpertMode";
      =     #Rapper.man_mode_locked;
      CALL  "FC21 Ventil 1A0-2E" (
           in_Ventil_Typ            := 0,
           in_Handbedienung_erlaubt := TRUE,
           in_Quitt_Stoerung_noetig := FALSE,
           in_Quitt_Stoerung        := TRUE,
           in_Anlage_ein            := #I_xSystemActive,
           in_Ansteuerung_Ventil    := #Rapper.auto_mode_control,
           in_Eingang_angesteuert   := FALSE,
           in_Eingang_nicht_angest  := FALSE,
           io_Ausgang_Ventil        := #q_xRepperValve,
           io_Ventil_in_Betrieb     := #Rapper.valve_in_operation,
           io_Stoerung              := #Rapper.fault,
           io_Ventilstruktur        := #Rapper);	// no feedback
NETWORK
TITLE = ------------------HOPPER'S STATES(REC/HP)-----------------------
NETWORK
TITLE = REC01 intern statuses(full, filled, empty)
      A     #INTERNAL.Flags.Switches.xHighLevelCovered;
      =     #INTERNAL.Flags.StatusREC.xFull;
//filled
      A     #SEQUENCES.Filling.RELEASE;
      A     #AngleValve.valve_in_operation;
      O     #INTERNAL.Flags.StatusREC.xFull;
      S     #INTERNAL.Flags.StatusREC.xFilled;
      A     #SEQUENCES.Discharging.RELEASE;
      A     #TIMERS.TON_DischargingTime.Q;
      A     #INTERNAL.Flags.xRequestPM;
      AN    #INTERNAL.Flags.StatusREC.xFull;
      O;
      A     #HMI.CMD.xSetEmpty;	// from VISU
      AN    #INTERNAL.Flags.StatusREC.xFull;
      AN    #SEQUENCES.Filling.ACTIVE;
      AN    #SEQUENCES.Filling.CLEANING;
      R     #INTERNAL.Flags.StatusREC.xFilled;
//empty
      AN    #INTERNAL.Flags.StatusREC.xFilled;
      =     #INTERNAL.Flags.StatusREC.xEmpty;
NETWORK
TITLE = -------------------LAMPS/TASTER LIGHTS--------------------------
NETWORK
TITLE = Traffic Lamps
// red 
      A     #SEQUENCES.Discharging.FAULTED;
      O;
      A(;
//    A     #IF_RECEIVER.CONTROL.CMD.Request
//   A     #IF_RECEIVER.CONTROL.CMD.FILL_Agg_FAULT
      O;
// A     #IF_RECEIVER.CONTROL.CMD.Request
// A     #IF_RECEIVER.CONTROL.CMD.DISCH_Agg_FAULT
      O;
//      A     #IF_RECEIVER.CONTROL.CMD.FILL_SEQ_FAULT
      );
//    O     #IF_RECEIVER.CONTROL.CMD.SFStop
//      =     #INTERNAL.Flags.BUTTONS_LAMPS.Red.Steady
//      A     #IF_RECEIVER.CONTROL.CMD.PressureFault
//      O     #IF_RECEIVER.CONTROL.CMD.SFStop
//      =     #INTERNAL.Flags.BUTTONS_LAMPS.Red.Flash
      CLR;
//      =     #INTERNAL.Flags.BUTTONS_LAMPS.Red.DoubleFlash
      CALL  "FC25 Lamp" (
           Steady                   := #INTERNAL.Flags.BUTTONS_LAMPS.Red.Steady,
           Flash                    := #INTERNAL.Flags.BUTTONS_LAMPS.Red.Flash,
           DoubleFlash              := #INTERNAL.Flags.BUTTONS_LAMPS.Red.DoubleFlash,
           LampTest                 := "GlobalLampTesting",
           Lamp                     := #q_xRedLamp);
//yellow
      CLR;
//      SET   
//      =     #INTERNAL.Flags.BUTTONS_LAMPS.Yellow.Steady
//      A     #IF_RECEIVER.CONTROL.CMD.Full
//      =     #INTERNAL.Flags.BUTTONS_LAMPS.Yellow.Flash
//      A     #fLowLevel
//      =     #INTERNAL.Flags.BUTTONS_LAMPS.Yellow.DoubleFlash
      CALL  "FC25 Lamp" (
           Steady                   := #INTERNAL.Flags.BUTTONS_LAMPS.Yellow.Steady,
           Flash                    := #INTERNAL.Flags.BUTTONS_LAMPS.Yellow.Flash,
           DoubleFlash              := #INTERNAL.Flags.BUTTONS_LAMPS.Yellow.DoubleFlash,
           LampTest                 := "GlobalLampTesting",
           Lamp                     := #q_xYellowLamp);
//green
//      A     #IF_RECEIVER.CONTROL.CMD.Request
      AN    #SEQUENCES.Discharging.FAULTED;
///      =     #INTERNAL.Flags.BUTTONS_LAMPS.Green.Steady
      A     #SEQUENCES.Discharging.ACTIVE;
//      =     #INTERNAL.Flags.BUTTONS_LAMPS.Green.Flash
      AN    #SEQUENCES.Discharging.ACTIVE;
      A     #SEQUENCES.Discharging.RELEASE;
//     =     #INTERNAL.Flags.BUTTONS_LAMPS.Green.DoubleFlash
      CALL  "FC25 Lamp" (
           Steady                   := #INTERNAL.Flags.BUTTONS_LAMPS.Green.Steady,
           Flash                    := #INTERNAL.Flags.BUTTONS_LAMPS.Green.Flash,
           DoubleFlash              := #INTERNAL.Flags.BUTTONS_LAMPS.Green.DoubleFlash,
           LampTest                 := "GlobalLampTesting",
           Lamp                     := #q_xGreenLamp);
NETWORK
TITLE = Discharging: FAULTED to STORAGE
      O     #f_xFullReceiver;
      O     #f_xNoStartConditions;
      =     #SEQUENCES.Discharging.FAULTED;
NETWORK
TITLE = ----------------------OUTPUT PFCs-------------------------------
NETWORK
TITLE = -------------------------STATUSES HMI---------------------------
NETWORK
TITLE = SEQ Status to HMI: Filling STATUS
      AN    #SEQUENCES.Filling.RELEASE;
      AN    #SEQUENCES.Filling.ACTIVE;
      AN    #SEQUENCES.Filling.CLEANING;
//      AN    #SEQUENCES.Filling.FAULTED
      JCN   FRA;	// status release assignment
      L     0;
      JU    FAF;	// status assignmnet is finished 
FRA:  A     #SEQUENCES.Filling.RELEASE;
      AN    #SEQUENCES.Filling.ACTIVE;
      AN    #SEQUENCES.Filling.CLEANING;
//      AN    #SEQUENCES.Filling.FAULTED
      JCN   FAA;	// status active 
      L     1;
      JU    FAF;
FAA:  A     #SEQUENCES.Filling.ACTIVE;
      AN    #SEQUENCES.Filling.CLEANING;
//      AN    #SEQUENCES.Filling.FAULTED
      JCN   FCA;
      L     2;
      JU    FAF;
FCA:  A     #SEQUENCES.Filling.CLEANING;
//      AN    #SEQUENCES.Filling.FAULTED
      JCN   FFA;
      L     3;
      JU    FAF;
FFA:  AN    #SEQUENCES.Filling.FAULTED;
      L     99;
FAF:  T     #HMI.PV.StatusFilling;
NETWORK
TITLE = Status to HMI: Discharging STATUS
      AN    #SEQUENCES.Discharging.RELEASE;
      AN    #SEQUENCES.Discharging.ACTIVE;
      AN    #SEQUENCES.Discharging.RESTDISCHARGE_REQ;
//     AN    #SEQUENCES.Discharging.RESTDISCHARGE_HP
//      AN    #SEQUENCES.Discharging.FAULTED
      JCN   DRA;	// status release assignment
      L     0;
      JU    DAF;	// status assignmnet is finished 
DRA:  A     #SEQUENCES.Discharging.RELEASE;	//released
      AN    #SEQUENCES.Discharging.ACTIVE;
      AN    #SEQUENCES.Discharging.RESTDISCHARGE_REQ;
      AN    #SEQUENCES.Discharging.reserve_1;
//      AN    #SEQUENCES.Discharging.FAULTED
      JCN   DAA;	// status active 
      L     1;
      JU    DAF;
DAA:  A     #SEQUENCES.Discharging.RELEASE;	//active
      A     #SEQUENCES.Discharging.ACTIVE;
      AN    #SEQUENCES.Discharging.RESTDISCHARGE_REQ;
      AN    #SEQUENCES.Discharging.reserve_1;
//      AN    #SEQUENCES.Discharging.FAULTED
      JCN   DAR1;
      L     2;
      JU    DAF;
DAR1: A     #SEQUENCES.Discharging.RESTDISCHARGE_REQ;	//rest discharge         rec01
      AN    #SEQUENCES.Discharging.reserve_1;
//      AN    #SEQUENCES.Discharging.FAULTED
      JCN   DAR2;
      L     3;
      JU    DAF;
DAR2: A     #SEQUENCES.Discharging.reserve_1;	//rest discharge hp
//      AN    #SEQUENCES.Discharging.FAULTED
      JCN   DAF;
      L     4;
      JU    DAF;
      A     #SEQUENCES.Discharging.FAULTED;
      L     99;
DAF:  T     #HMI.PV.StatusDischarging;
NETWORK
TITLE = Statuses to HMI for REC01 and HP01 
//REC01
      A     #INTERNAL.Flags.StatusREC.xEmpty;
      JCN   HS1;	// hopper status
      L     1;
      JU    HSE;	// hopper state end
HS1:  A     #INTERNAL.Flags.StatusREC.xFull;
      JCN   HS2;
      L     2;
      JU    HSE;
HS2:  A     #INTERNAL.Flags.StatusREC.xFilled;
      JCN   HS3;
      L     3;
      JU    HSE;
HS3:  L     0;
HSE:  T     #HMI.PV.StatusREC01;
NETWORK
TITLE = Status to HMI: PFC to/from Packaging Machine
// 
//      A     #iPFCPM_Ready
//      =     #HMI.STATE.PM_Ready
// from Packaging 
//      A     #iPFCPM_Request
//      =     #HMI.STATE.PFC_Request
// to Packaging
//      A     #qPFCPM_Product
//      =     #HMI.STATE.Product_PM
//      A     #qPFCPM_Active
//      =     #HMI.STATE.Active_PM
//      AN    #iPFCPM_Request
//      =     #fNoPFCRequest
NETWORK
TITLE = ------------Resetting----------------
NETWORK
TITLE = Reset Recipe???? (is not needed)
NETWORK
TITLE = -----------------------INTERFACES-------------------------------
NETWORK
TITLE = Storage location
      L     #I_iIFStoLocParDB;
      T     #INTERNAL.IF.Storage.StorageLocation_DB;
      L     #I_iIFStorageDW;
      T     #INTERNAL.IF.Storage.StorageLocation_DW;
      SET;
      =     #IF_Storage.CONTROL.CMD.xConnect;
      CALL  "FC40 copy Obj-SST Master" (
           i_Freigabe               := #IF_Storage.CONTROL.CMD.xConnect,
           i_Ziel_DB                := #INTERNAL.IF.Storage.StorageLocation_DB,
           i_Ziel_DW                := #INTERNAL.IF.Storage.StorageLocation_DW,
           i_SST_von_Ziel           := #IF_Storage.STATUS,
           i_SST_an_Ziel            := #IF_Storage.CONTROL,
           Ziel_frei                := #INTERNAL.IF.Storage.IF_Silo_free);
      NOP   0;
NETWORK
TITLE = Blower
      L     #I_iIFVacuumPumpDB;
      T     #INTERNAL.IF.Blower.Blower_DB;
      L     #I_iIFVacuumPumpDW;
      T     #INTERNAL.IF.Blower.Blower_DW;
      CALL  "FC40 copy Obj-SST Master" (
           i_Freigabe               := #IF_VP.CONTROL.CMD.xRequest,
           i_Ziel_DB                := #INTERNAL.IF.Blower.Blower_DB,
           i_Ziel_DW                := #INTERNAL.IF.Blower.Blower_DW,
           i_SST_von_Ziel           := #IF_VP.STATUS,
           i_SST_an_Ziel            := #IF_VP.CONTROL,
           Ziel_frei                := #INTERNAL.IF.Blower.Blower_free);
END_FUNCTION_BLOCK

FUNCTION_BLOCK "VACUUM PUMP"	// FB 1051
TITLE = Blower PMP01
//Creation:
//Date:            Author:                                               Version
//--------------------------------------------------------------------------------
//29.03.2018     ilia                                   01.00.00
//
//Changes:
//No. Date:        Who       Description                           Mark   Version 
//--------------------------------------------------------------------------------
//01
//________________________________________________________________________________
//Function:
//1. Maximum 6 switching cycles per hour ' 10 minutes restart protection time
//
AUTHOR : ilia
NAME : project
VERSION : 1.0
VAR_INPUT
  IF_VP1_FC_DB : INT ;
  IF_VP1_FC_DW : INT ;
  i_piwPressureVP1 : INT ;	//analogue input address
  i_xFAValveClose : BOOL ;
  i_xFAValveOpen : BOOL ;
  i_xSystemActive : BOOL ;	//system control on
  ack_xFAValve : BOOL ;
  ack_OverPressureVP1 : BOOL ;
END_VAR
VAR_IN_OUT
  q_xFAValve : BOOL ;
  f_xFAValve : BOOL ;
  f_xPressureFaultVP1 : BOOL ;
  f_xBrokenWirePTVPV1 : BOOL ;
  f_xParErrorPTVPVP1 : BOOL ;
END_VAR
VAR
  reserve_IO : ARRAY  [10 .. 49 ] OF BYTE ;
  HMI : STRUCT 	//Interface of HMI
   CMD : STRUCT
    reserve : BOOL ;
    reserve_1 : BOOL ;
    reserve_2 : BOOL ;
    reserve_3 : BOOL ;
    reserve_4 : BOOL ;
    reserve_5 : BOOL ;
    reserve_6 : BOOL ;
    reserve_7 : BOOL ;
    reserve_8 : BOOL ;
    reserve_9 : BOOL ;
    reserve_10 : BOOL ;
    reserve_11 : BOOL ;
    reserve_12 : BOOL ;
    reserve_13 : BOOL ;
    reserve_14 : BOOL ;
    reserve_15 : BOOL ;
   END_STRUCT ;
   STATE : STRUCT
    xxPressureFault : BOOL ;
    xxEmtyPressure : BOOL ;
    VP1Locked : BOOL ;
    reserve_4 : BOOL ;
    reserve_5 : BOOL ;
    reserve_6 : BOOL ;
    reserve_7 : BOOL ;
    reserve_8 : BOOL ;
    reserve_9 : BOOL ;
    reserve_10 : BOOL ;
    reserve_11 : BOOL ;
    reserve_12 : BOOL ;
    reserve_13 : BOOL ;
    reserve : BOOL ;
   END_STRUCT ;
   PARAM : STRUCT
    VPOffDelayTime : REAL  := 6.000000e+001;
    res : REAL ;
    res_1 : REAL ;
    res_2 : REAL ;
    res_3 : REAL ;
    HDDelayOn : REAL  := 2.000000e+000;
    reserve_2 : REAL ;
    reserve_3 : REAL ;
    reserve_4 : REAL ;
    SF_set_cycles : INT  := 6;
    reserve_6 : INT ;
    reserve_7 : INT ;
    reserve_8 : INT ;
    reserve_9 : INT ;
    reserve_10 : INT ;
   END_STRUCT ;
   PV : STRUCT
    BlowerOffDelayTime : REAL ;
    res : REAL ;
    res_1 : REAL ;
    res_2 : REAL ;
    res_3 : REAL ;
    res_4 : REAL ;
    HoseDiverterDelayOn : REAL ;
    reserve_4 : REAL ;
    RestartIntervalVP1 : REAL ;
    SF_act_Cycles : INT ;
    SF_Status : INT ;
    reserve_8 : INT ;
    reserve_9 : INT ;
    reserve_10 : INT ;
    reserve_11 : INT ;
   END_STRUCT ;
  END_STRUCT ;
  PROD : STRUCT 	//Interface of Production
   FROM : STRUCT
    reserve : INT ;
    reserve_1 : INT ;
    reserve_2 : INT ;
    reserve_3 : INT ;
    reserve_4 : INT ;
    reserve_5 : REAL ;
    reserve_6 : REAL ;
    CMD : STRUCT
     reserve : BOOL ;
     reserve_1 : BOOL ;
     reserve_2 : BOOL ;
     reserve_3 : BOOL ;
     reserve_4 : BOOL ;
     reserve_5 : BOOL ;
     reserve_6 : BOOL ;
     reserve_7 : BOOL ;
     reserve_8 : BOOL ;
     reserve_9 : BOOL ;
     reserve_10 : BOOL ;
     reserve_11 : BOOL ;
     reserve_12 : BOOL ;
     reserve_13 : BOOL ;
     reserve_14 : BOOL ;
     reserve_15 : BOOL ;
    END_STRUCT ;
   END_STRUCT ;
   TO : STRUCT
    reserve : INT ;
    reserve_1 : INT ;
    reserve_2 : INT ;
    reserve_3 : INT ;
    reserve_4 : INT ;
    reserve_5 : REAL ;
    reserve_6 : REAL ;
    STATE : STRUCT
     reserve : BOOL ;
     reserve_1 : BOOL ;
     reserve_2 : BOOL ;
     reserve_3 : BOOL ;
     reserve_4 : BOOL ;
     reserve_5 : BOOL ;
     reserve_6 : BOOL ;
     reserve_7 : BOOL ;
     reserve_8 : BOOL ;
     reserve_9 : BOOL ;
     reserve_10 : BOOL ;
     reserve_11 : BOOL ;
     reserve_12 : BOOL ;
     reserve_13 : BOOL ;
     reserve_14 : BOOL ;
     reserve_15 : BOOL ;
    END_STRUCT ;
   END_STRUCT ;
   reserve : ARRAY  [40 .. 49 ] OF BYTE ;
  END_STRUCT ;
  IF_Consumer : STRUCT 	//Interface Blower in blower object
   CONTROL : STRUCT
    Answer_DB : INT ;
    Answer_DW : INT ;
    SpeedVP1 : INT ;
    NumberOfPumps : INT ;
    reserve_3 : INT ;
    reserve_4 : REAL ;
    reserve_5 : REAL ;
    CMD : STRUCT
     Request : BOOL ;
     Release : BOOL ;
     reserve : BOOL ;
     reserve_1 : BOOL ;
     reserve_2 : BOOL ;
     reserve_3 : BOOL ;
     reserve_4 : BOOL ;
     reserve_5 : BOOL ;
     reserve_6 : BOOL ;
     reserve_7 : BOOL ;
     reserve_8 : BOOL ;
     reserve_9 : BOOL ;
     reserve_10 : BOOL ;
     reserve_11 : BOOL ;
     reserve_12 : BOOL ;
     reserve_13 : BOOL ;
    END_STRUCT ;
   END_STRUCT ;
   STATUS : STRUCT
    reserve_1 : INT ;
    reserve_2 : INT ;
    reserve_3 : INT ;
    reserve_4 : INT ;
    reserve_5 : INT ;
    ActualPressure : REAL ;
    reserve_6 : REAL ;
    STATE : STRUCT
     Ready : BOOL ;
     Active : BOOL ;
     PressureFault : BOOL ;
     EmptyPressurReached : BOOL ;
     Fault : BOOL ;
     SF_Full : BOOL ;
     reserve_2 : BOOL ;
     reserve_3 : BOOL ;
     reserve_4 : BOOL ;
     reserve_5 : BOOL ;
     reserve_6 : BOOL ;
     reserve_7 : BOOL ;
     reserve_8 : BOOL ;
     reserve_9 : BOOL ;
     reserve_10 : BOOL ;
     reserve_11 : BOOL ;
    END_STRUCT ;
   END_STRUCT ;
  END_STRUCT ;
  IF_FC_VP1 : STRUCT 	//Interface FC in active object
   STATUS : STRUCT
    ActualFrequency : REAL ;
    reserve : INT ;
    reserve_1 : INT ;
    reserve_2 : INT ;
    reserve_3 : INT ;
    reserve_4 : INT ;
    reserve_5 : REAL ;
    STATE : STRUCT
     Ready : BOOL ;
     Active : BOOL ;
     Fault : BOOL ;
     reserve : BOOL ;
     reserve_1 : BOOL ;
     reserve_2 : BOOL ;
     reserve_3 : BOOL ;
     reserve_4 : BOOL ;
     reserve_5 : BOOL ;
     reserve_6 : BOOL ;
     reserve_7 : BOOL ;
     reserve_8 : BOOL ;
     reserve_9 : BOOL ;
     reserve_10 : BOOL ;
     reserve_11 : BOOL ;
     reserve_12 : BOOL ;
    END_STRUCT ;
   END_STRUCT ;
   CONTROL : STRUCT
    Answer_DB : INT ;
    Answer_DW : INT ;
    Frequency_Set : REAL ;
    No_motor_data : INT ;
    reserve : INT ;
    reserve_1 : INT ;
    reserve_2 : REAL ;
    CMD : STRUCT
     Request : BOOL ;
     Release : BOOL ;
     Left_run : BOOL ;
     reserve : BOOL ;
     reserve_1 : BOOL ;
     reserve_2 : BOOL ;
     reserve_3 : BOOL ;
     reserve_4 : BOOL ;
     reserve_5 : BOOL ;
     reserve_6 : BOOL ;
     reserve_7 : BOOL ;
     reserve_8 : BOOL ;
     reserve_9 : BOOL ;
     reserve_10 : BOOL ;
     reserve_11 : BOOL ;
     reserve_12 : BOOL ;
    END_STRUCT ;
   END_STRUCT ;
  END_STRUCT ;
  reserve_IF : ARRAY  [280 .. 499 ] OF BYTE ;
  VP1 : STRUCT 	//motor object
   parameter : STRUCT
    motor_on : BOOL  := TRUE;	//activate motor structure
    clock_on : BOOL ;	//activate clock structure
    FC_on : BOOL  := TRUE;	//activate frequency converter structure
    hour_meter_on : BOOL ;	//activate hour meter
    reserve_4 : BOOL ;
    reserve_5 : BOOL ;
    reserve_6 : BOOL ;
    reserve_7 : BOOL ;
   END_STRUCT ;
   quit_motor : BOOL ;	//1 = quit motor on
   input_motor : BOOL ;	//1 = input motor on (return indication)
   motor_locked : BOOL ;	//1 = motor locked (in manual and auto mode) e.g. repair-/safety switch
   auto_mode_control : BOOL ;	//1 = release/control of motor in auto mode
   motor_in_operation : BOOL ;	//1 = signal motor in operation
   fault : BOOL ;	//1 = signal motor fault
   man_mode_to_SCADA : BOOL ;	//0 = Automatik Mode, 1 = Hand Mode
   man_mode_from_SCADA : BOOL ;	//0 = Automatik Mode, 1 = Hand Mode
   man_mode_control : BOOL ;	//1 = release/control of motor in manual mode (from SCADA)
   man_mode_locked : BOOL ;	//1 = change to manual mode locked, motor is in automatic use
   start_with_impulse : BOOL  := TRUE;	//1 = start cycle with impulse
   set_cycles_reached : BOOL ;	//1 = set number of cycles has been reached
   continous_clock : BOOL  := TRUE;	//1 = continous clock / 0 = set number of clocks
   simulation : BOOL ;	//1 = simulation of object
   release_clock : BOOL ;	//1 = release bit for clock FC
   quit_clock : BOOL ;	//quit for clock FC, if release_clock = TRUE
   set_time_fault : INT  := 5;	//fault evaluation time in seconds
   actual_time_fault : INT ;	//actual fault evaluation time in seconds
   impulse_time : REAL  := 5.000000e+000;	//impulse time for clock in seconds
   break_time : REAL  := 5.000000e+000;	//break time for clock in seconds
   time_counter : REAL ;	//time counter (elapsed time)
   set_cycles : INT ;	//number of clocks if not continous clock
   clock_counter : INT ;	//clock counter
   FCs : STRUCT 	//frequency converter
    FC_in_operation : BOOL ;	//1 = FU in Betrieb
    fault : BOOL ;	//1 = FC fault
    set_revolutions_man_mode : INT  := 200;	//revolutions in permille in manual mode
    actual_revolutions : INT ;	//actual revolutions FC in man/auto mode
   END_STRUCT ;
   hour_meter : STRUCT 	//hour meter
    reset : BOOL ;	//reset hour meter
    warning : BOOL ;	//warning time exceeded
    alarm : BOOL ;	//alarm time exceeded
    actual_operating_hours : REAL ;	//actual operating hours (in hours)
    set_time_warning : REAL ;	//set time for warning (in hours)
    set_time_alarm : REAL ;	//set time for alarm (in hours)
    second_counter_oh : INT ;	//seconds of the actual operatin hours
   END_STRUCT ;
   system_on : BOOL ;	//system released resepectively system area released after emergency stopping
   object_state : INT ;	//1=grey; 5=green; 9=white; 15=yellow; 16=red
  END_STRUCT ;
  FAValve : STRUCT 	//Fresh Aur Valve object with 1Q and 0-2I
   parameter : STRUCT
    valve_on : BOOL  := TRUE;	//activate valve structure
    clock_on : BOOL ;	//activate clock structure
    reserve_3 : BOOL ;
    switching_number_on : BOOL ;	//activate switching number counter
    reserve_4 : BOOL ;
    parameter_1Q : BOOL ;	//valve type with 1 quit 0 inputs
    parameter_1Q_1I : BOOL ;	//valve type with 1 quit 1 input (=)
    parameter_1Q_1IN : BOOL ;	//valve type with 1 quit 1 input (<>)
    parameter_1Q_2I : BOOL  := TRUE;	//valve type with 1 quit 2 inputs
    parameter_text_pos_1 : BOOL ;
    parameter_text_straight : BOOL ;
    parameter_text_inverse : BOOL ;	//select text inverse = "close/open" or "bypass/convey" aso.
    parameter_text_open : BOOL ;	//select text quit = "open/close"
    parameter_text_convey : BOOL  := TRUE;	//select text quit = "convey/bypass"
    parameter_text_on : BOOL ;	//select text quit = "on/off"
    parameter_text_up : BOOL ;	//select text quit = "up/down"
   END_STRUCT ;
   quit_valve : BOOL ;	//1 = quit valve
   input_valve_set : BOOL ;	//1 = input valve, if quit valve set
   input_valve_not_set : BOOL ;	//1 = input valve, if quit valve not set
   auto_mode_control : BOOL ;	//1 = release/control of valve in auto mode
   valve_in_operation : BOOL ;	//1 = signal valve in operation
   fault : BOOL ;	//1 = signal valve fault
   man_mode_to_SCADA : BOOL ;	//0 = automatic mode , 1 = manual mode
   man_mode_from_SCADA : BOOL ;	//0 = automatic mode , 1 = manual mode
   man_mode_control : BOOL ;	//1 = release/control of valve in manual mode (from SCADA)
   man_mode_locked : BOOL ;	//1 = change to manual mode locked, valve is in automatic use
   start_with_impulse : BOOL ;	//1 = start cycle with impluse
   set_cycles_reached : BOOL ;	//1 = set number of cycles has been reached
   continous_clock : BOOL ;	//1 = continous clock / 0 = set number of clocks
   simulation : BOOL ;	//1 = simulation of object
   release_clock : BOOL ;	//1 = release bit for clock FC
   quit_clock : BOOL ;	//quit for clock FC, if release_clock = TRUE
   set_time_fault : INT  := 5;	//fault evaluation time in seconds
   actual_time_fault : INT ;	//actual fault evaluation time in seconds
   impulse_time : REAL  := 5.000000e+000;	//impulse time for clock in seconds
   break_time : REAL  := 5.000000e+000;	//break time for clock in seconds
   time_counter : REAL ;	//time counter (elapsed time)
   set_cycles : INT ;	//number of clocks if not continous clock
   clock_counter : INT ;	//clock counter
   switching_number_counter : STRUCT 	//switching number counter
    reset : BOOL ;	//reset switching number counter
    warning : BOOL ;	//warning number exceeded
    alarm : BOOL ;	//alarm number exceeded
    flank_flag : BOOL ;	//internal flag
    actual_switching_number : REAL ;	//actual switching number
    set_number_warning : REAL ;	//set number for warning
    set_number_alarm : REAL ;	//set number for alarm
   END_STRUCT ;
   set_time_in_operation : INT ;	//1IoO: set time for delay of "valve in operation"
   real_time_in_operation : INT ;	//1IoO: real time for delay of "valve in operation"
   system_on : BOOL ;	//system released resepectively system area released after emergency stopping
   reserve : ARRAY  [44 .. 47 ] OF BYTE ;
   object_state : INT ;	//1=grey; 5=green; 9=white; 15=yellow; 16=red
  END_STRUCT ;
  reserve_Cmod : ARRAY  [600 .. 999 ] OF BYTE ;
  PressureVP1 : STRUCT
   parameters : STRUCT
    pressureAIOn : BOOL  := TRUE;
    reserve1 : BOOL ;
    reserve2 : BOOL ;
    CounterOverPressure : BOOL  := TRUE;
    CounterEmptyPressure : BOOL ;
    CounterActivePressure : BOOL ;
    reserve_6 : BOOL ;
    reserve_7 : BOOL ;
    OverPressure : BOOL  := TRUE;
    EmptyPressure : BOOL  := TRUE;
    ActivePressure : BOOL  := TRUE;
    reserve_13 : BOOL ;
    ManOpSimEn : BOOL  := TRUE;
    ManOpAdjustEn : BOOL  := TRUE;
    reserve_14 : BOOL ;
    reserve_15 : BOOL ;
    uom_code : INT ;
   END_STRUCT ;
   ManModeAct : BOOL ;
   ManModeOp : BOOL ;
   ManModeLock : BOOL ;
   ManOpPressureEmpty : BOOL ;
   ManOpPressureConveying : BOOL ;
   ManOpPressureAlarm : BOOL ;
   ManOpPressureAdjust : BOOL ;
   SystemOn : BOOL ;
   ScalingErr : BOOL ;
   OVErr : BOOL ;
   ParErr : BOOL ;
   fOverPressure : BOOL ;
   fOverPressureEn : BOOL ;
   fOverPressureAck : BOOL ;
   Overpressure : BOOL ;
   EmptyPressure : BOOL ;
   ActivePressure : BOOL ;
   Active : BOOL ;
   AdjustRelease : BOOL ;
   AdjustPulse : BOOL ;
   ManAdjustReq : BOOL ;
   ManAdjustRdy : BOOL ;
   CounterReset : BOOL ;
   CounterEdge : BOOL ;
   PVAct : REAL ;
   PressureOffset : REAL ;
   MaxOverPressurePV : REAL  := -6.000000e+002;
   MinOverPressurePV : REAL  := -3.000000e+002;
   EmptyPressurePV : REAL  := -2.000000e+002;
   ActivePressurePV : REAL ;
   EmptyDelay : INT  := 5;
   ActiveDelay : INT  := 5;
   AlarmDelay : INT  := 10;
   EmptyDelayCounter : INT ;
   ActiveDelayCounter : INT ;
   AlarmDelayCounter : INT ;
   CounterAct : REAL ;
   object_state : INT ;
  END_STRUCT ;
  reserve_Binary : ARRAY  [1050 .. 1499 ] OF BYTE ;
  TIMES : STRUCT 	//ten timers
   TOF_DelayVP : STRUCT
    IN : BOOL ;
    RST : BOOL ;
    IMP : BOOL ;
    Q : BOOL ;
    PT : REAL ;
    ET : REAL ;
   END_STRUCT ;
   TOF_RestartProtectVP1 : STRUCT
    IN : BOOL ;
    RST : BOOL ;
    IMP : BOOL ;
    Q : BOOL ;
    PT : REAL ;
    ET : REAL ;
   END_STRUCT ;
   TOF_RestartProtectVP2 : STRUCT
    IN : BOOL ;
    RST : BOOL ;
    IMP : BOOL ;
    Q : BOOL ;
    PT : REAL ;
    ET : REAL ;
   END_STRUCT ;
   TON_HoseDiverter : STRUCT
    IN : BOOL ;
    RST : BOOL ;
    IMP : BOOL ;
    Q : BOOL ;
    PT : REAL  := 2.000000e+000;
    ET : REAL ;
   END_STRUCT ;
   TON_Start_VP2 : STRUCT
    IN : BOOL ;
    RST : BOOL ;
    IMP : BOOL ;
    Q : BOOL ;
    PT : REAL ;
    ET : REAL ;
   END_STRUCT ;
   TOF_HoseDiverter : STRUCT
    IN : BOOL ;
    RST : BOOL ;
    IMP : BOOL ;
    Q : BOOL ;
    PT : REAL ;
    ET : REAL ;
   END_STRUCT ;
   reserve_3 : STRUCT
    IN : BOOL ;
    RST : BOOL ;
    IMP : BOOL ;
    Q : BOOL ;
    PT : REAL ;
    ET : REAL ;
   END_STRUCT ;
   reserve_4 : STRUCT
    IN : BOOL ;
    RST : BOOL ;
    IMP : BOOL ;
    Q : BOOL ;
    PT : REAL ;
    ET : REAL ;
   END_STRUCT ;
   reserve_5 : STRUCT
    IN : BOOL ;
    RST : BOOL ;
    IMP : BOOL ;
    Q : BOOL ;
    PT : REAL ;
    ET : REAL ;
   END_STRUCT ;
   reserve_6 : STRUCT
    IN : BOOL ;
    RST : BOOL ;
    IMP : BOOL ;
    Q : BOOL ;
    PT : REAL ;
    ET : REAL ;
   END_STRUCT ;
  END_STRUCT ;
  SEQUENCES : STRUCT
   Sequence : STRUCT
    AUTO : BOOL ;
    MANUAL : BOOL ;
    LOCKED : BOOL ;
    RELEASE : BOOL ;
    ACTIVE : BOOL ;
    reserve_2 : BOOL ;
    reserve_3 : BOOL ;
    reserve_4 : BOOL ;
    reserve_5 : BOOL ;
    reserve_6 : BOOL ;
    reserve_7 : BOOL ;
    reserve_8 : BOOL ;
    reserve_9 : BOOL ;
    reserve_10 : BOOL ;
    reserve_11 : BOOL ;
    reserve_12 : BOOL ;
   END_STRUCT ;
   reserve : ARRAY  [2 .. 99 ] OF BYTE ;
  END_STRUCT ;
  INTERNAL : STRUCT
   IF : STRUCT
    VacuumPump : STRUCT
     VP1_FaultControl : BOOL ;
     VP2_FaultControl : BOOL ;
     reserve : BOOL ;
     reserve_2 : BOOL ;
     reserve_3 : BOOL ;
     reserve_4 : BOOL ;
     reserve_5 : BOOL ;
     reserve_5_1 : BOOL ;
     SpeedVP1_PARAM : INT ;
     SpeedVP1_PV : REAL ;
    END_STRUCT ;
    SF01 : STRUCT
     HighLevelSF_FaultControl : BOOL ;
     ManFlapSF_FaultControl : BOOL ;
     SF_ready : BOOL ;
     CleaningFilterAfterSeq : BOOL ;
     reserve : BOOL ;
     resrve : BOOL ;
     res : BOOL ;
     res_1 : BOOL ;
     res_2 : INT ;
     res_3 : REAL ;
    END_STRUCT ;
    VP_FC : STRUCT
     free : BOOL ;
     res_2 : BOOL ;
     res_3 : BOOL ;
     res_4 : BOOL ;
     reserve : BOOL ;
     resrve : BOOL ;
     res : BOOL ;
     res_1 : BOOL ;
    END_STRUCT ;
    reserve_6 : BOOL ;
    reserve_7 : BOOL ;
    reserve_8 : BOOL ;
    reserve_9 : BOOL ;
    reserve_10 : BOOL ;
    reserve_11 : BOOL ;
    reserve_12 : BOOL ;
    reserve_13 : BOOL ;
    reserve_14 : BOOL ;
    reserve_15 : BOOL ;
   END_STRUCT ;
   Flags : STRUCT
    BinaryObjects : STRUCT
     Res : BOOL ;
     Res_1 : BOOL ;
     RES_2 : BOOL ;
     RES_3 : BOOL ;
     RES_4 : BOOL ;
     RES_5 : BOOL ;
     RES_6 : BOOL ;
     RES_7 : BOOL ;
    END_STRUCT ;
    FP_VP1_ON : STRUCT
     help : BOOL ;
     pulse : BOOL ;
    END_STRUCT ;
    Res_1 : STRUCT
     help : BOOL ;
     pulse : BOOL ;
    END_STRUCT ;
    FN_SequenceActive : STRUCT
     help : BOOL ;
     pulse : BOOL ;
    END_STRUCT ;
    FP_reserve : STRUCT
     help : BOOL ;
     pulse : BOOL ;
    END_STRUCT ;
    reserve_3 : BOOL ;
    reserve_4 : BOOL ;
    reserve_5 : BOOL ;
    reserve_6 : BOOL ;
    reserve_7 : BOOL ;
    reserve_8 : BOOL ;
    reserve_9 : BOOL ;
    reserve_10 : BOOL ;
   END_STRUCT ;
   PressureTransmitter : STRUCT
    Analog : STRUCT
     in : STRUCT
      UperLimit : REAL  := 1.000000e+003;	//Uper limit analog value
      LowerLimit : REAL  := -1.000000e+003;	//Lower limit analog value
      MaxDigit : REAL  := 2.764800e+004;	//Uper limit analog channel
      MinDigit : REAL ;	//Lower limit analog channel
      Simulation : BOOL ;	//Simulation = 1
      DB_Simulation_IO : INT  := 92;	//DB for simulation
     END_STRUCT ;
     out : STRUCT
      Value : REAL ;	//IO Analog value
      Broken_wire : BOOL ;	//Fault broken wire
      Reserve : INT ;
     END_STRUCT ;
    END_STRUCT ;
    Evaluation : STRUCT
     in : STRUCT
      Delay_Adjust : REAL  := 1.000000e+001;	//Delay adjust of Pressure Transmitter
      Selection_S_D : CHAR  := 'S';	//Selection suction-/pressure conveying ('S' or 'D')
      REL_Pressure_fault : BOOL  := TRUE;	//Release Pressure fault
      Time_counter : REAL ;	//Time counter delay adjust
      Output_Timer : BOOL ;	//Timer output delay adjust
     END_STRUCT ;
     out : STRUCT
      Relative_Pressure : REAL ;	//Relative Pressure
      Memory_Pressure : REAL ;	//Memory Pressure
      Pressure_fault_active : BOOL ;	//Pressure fault
      Empty_Pressure_reached : BOOL ;	//Below Empty Pressure
      output_delay_calibration : BOOL ;
     END_STRUCT ;
    END_STRUCT ;
   END_STRUCT ;
   Instance_DB_number : INT ;
   RestartProtectTime : REAL ;
  END_STRUCT ;
END_VAR
VAR_TEMP
  dummyBool : BOOL ;
END_VAR
BEGIN
NETWORK
TITLE = ---- instance DB ----
      L     0;
      L     DINO;
      ==I;
      BEC;
      T     #INTERNAL.Instance_DB_number;
NETWORK
TITLE = ----------------SEQUENCES AUTO/LOCKED/MANUAL-----------------
NETWORK
TITLE =  Sequence AUTO
      AN    #SEQUENCES.Sequence.LOCKED;
      =     #SEQUENCES.Sequence.AUTO;
NETWORK
TITLE =  Sequence Manual
      O     #VP1.man_mode_to_SCADA;
      O     #FAValve.man_mode_to_SCADA;
      =     #SEQUENCES.Sequence.MANUAL;
NETWORK
TITLE =  Sequence Locked
//BLOCK VP ALSO??????
      A     #SEQUENCES.Sequence.MANUAL;
      ON    #i_xSystemActive;
// MUST BE BLOCK VP 
      =     #SEQUENCES.Sequence.LOCKED;
NETWORK
TITLE = ---------------------SENSORS/SWITCHES --------------------------
NETWORK
TITLE = ------------------PRESSURE TRANSMITTERS-------------------------
NETWORK
TITLE = PressureTransmitter VP01
      L     -5.000000e+00;	// 2.000000e+001 
      T     #PressureVP1.ActivePressurePV;
      CALL  "PressureAi" (
           ManOpEn                  := TRUE,
           ManModeTrack             := TRUE,
           NegEvalEn                := TRUE,
           OVErrEn                  := TRUE,
           AlarmOprEn               := TRUE,
           AlarmOprAckEn            := FALSE,
           DigitMin                 := 0,
           DigitMax                 := 27648,
           ValueMin                 := -1.000000e+03,
           ValueMax                 := 1.000000e+03,
           ValueSubs                := 1.000000e+01,
           Configuration            := W#16#0,
           UOM                      := 1138,
           iSystemOn                := #i_xSystemActive,
           iwDigit                  := #i_piwPressureVP1,
           iActive                  := #PressureVP1.Active,
           aAlarmOprAck             := #ack_OverPressureVP1,
           PVAct                    := #PressureVP1.PVAct,
           fAlarmOpr                := #PressureVP1.fOverPressure,
           OverPressure             := #PressureVP1.Overpressure,
           EmptyPressure            := #PressureVP1.EmptyPressure,
           ActivePressure           := #PressureVP1.ActivePressure,
           fScalingErr              := #PressureVP1.ScalingErr,
           fOVErr                   := #PressureVP1.OVErr,
           fParErr                  := #f_xParErrorPTVPVP1,
           ioStructure              := #PressureVP1);	//mbar / #fPressureFault
      A     #PressureVP1.fOverPressure;	// #PressureTransmittter.Overpressure
      =     #f_xPressureFaultVP1;
      A     #PressureVP1.OVErr;
      =     #f_xBrokenWirePTVPV1;
NETWORK
TITLE = -----------------------------SEQUENCES--------------------------
NETWORK
TITLE = Sequence: ready to consumer
      A     #SEQUENCES.Sequence.AUTO;
      A     #IF_Consumer.CONTROL.CMD.Request;
      AN    #f_xFAValve;
      =     #IF_Consumer.STATUS.STATE.Ready;
NETWORK
TITLE = Sequence: release vacuum pump (VP1)
//blower off delay
      A     #SEQUENCES.Sequence.AUTO;
      A     #IF_Consumer.CONTROL.CMD.Request;
      A     #IF_Consumer.STATUS.STATE.Ready;
      A     #IF_Consumer.CONTROL.CMD.Release;
      =     #TIMES.TOF_DelayVP.IN;
      ON    #i_xSystemActive;
      =     #TIMES.TOF_DelayVP.RST;
      CALL  "FC3 Timernachbildung" (
           in_Freigabe              := #TIMES.TOF_DelayVP.IN,
           in_Reset                 := #TIMES.TOF_DelayVP.RST,
           in_Impuls                := "M1.7 ClockTimerFunction",
           in_Impulszeit_in_100ms   := "MW 6 Timer Val Cycle FCs",
           in_Verzoegerungsart      := B#16#41,
           in_Verzoegerungszeit     := #HMI.PARAM.VPOffDelayTime,
           io_Ausgangssignal        := #TIMES.TOF_DelayVP.Q,
           io_Zeitzaehler           := #TIMES.TOF_DelayVP.ET);
      L     #TIMES.TOF_DelayVP.ET;
      T     #HMI.PV.BlowerOffDelayTime;
      A     #TIMES.TOF_DelayVP.Q;
      =     #VP1.auto_mode_control;
NETWORK
TITLE = Sequence: release VP1 - with frequency Converter
//FC request
      A     #SEQUENCES.Sequence.AUTO;
      A     #IF_Consumer.CONTROL.CMD.Request;
      A     #IF_Consumer.STATUS.STATE.Ready;
      O;
      A     #VP1.man_mode_to_SCADA;
      A     #VP1.man_mode_control;
      O;
      A     #IF_FC_VP1.STATUS.STATE.Active;
      =     #IF_FC_VP1.CONTROL.CMD.Request;
      A     #TIMES.TOF_RestartProtectVP1.Q;
      AN    #VP1.motor_in_operation;
      O;
      AN    #IF_FC_VP1.STATUS.STATE.Ready;
      A     #IF_FC_VP1.CONTROL.CMD.Request;
      O;
      A     #IF_FC_VP1.STATUS.STATE.Fault;
      =     #VP1.motor_locked;
      A     #VP1.quit_motor;
      =     #VP1.input_motor;
      CALL  "FC20 Motor 1A1E" (
           in_Handbedienung_erlaubt := TRUE,
           in_Quitt_Stoerung_noetig := TRUE,
           in_Anlage_ein            := #i_xSystemActive,
           in_Quitt_Stoerung        := #dummyBool,
           in_Ansteuerung_Motor     := #VP1.auto_mode_control,
           in_Eingang_Motor         := #VP1.input_motor,
           io_Ausgang_Motor         := #VP1.quit_motor,
           io_Motor_in_Betrieb      := #VP1.motor_in_operation,
           io_Stoerung              := #VP1.fault,
           io_Motorstruktur         := #VP1);
//FC release
      A(;
      A     #VP1.auto_mode_control;
      O;
      A     #VP1.man_mode_to_SCADA;
      A     #VP1.man_mode_control;
      );
      A     #IF_FC_VP1.CONTROL.CMD.Request;
      A     #IF_FC_VP1.STATUS.STATE.Ready;
      A     #VP1.motor_in_operation;
      =     #IF_FC_VP1.CONTROL.CMD.Release;
NETWORK
TITLE = Sequence: frequency to/from FC VP1
      A     #VP1.man_mode_to_SCADA;
      A     #VP1.man_mode_control;
      L     #IF_Consumer.CONTROL.SpeedVP1;
      JCN   VNM;	// man mode 
      L     #VP1.FCs.set_revolutions_man_mode;
      L     10;
      /I;
VNM:  T     #INTERNAL.IF.VacuumPump.SpeedVP1_PARAM;
// to FC
      L     #INTERNAL.IF.VacuumPump.SpeedVP1_PARAM;
      ITD;
      DTR;
      T     #IF_FC_VP1.CONTROL.Frequency_Set;
//from FC
      L     #IF_FC_VP1.STATUS.ActualFrequency;
      T     #INTERNAL.IF.VacuumPump.SpeedVP1_PV;
      A     #VP1.man_mode_to_SCADA;
      A     #VP1.man_mode_control;
      L     0;
      JCN   VNM1;
      L     #INTERNAL.IF.VacuumPump.SpeedVP1_PV;
      RND;
      L     10;
      *I;
VNM1: T     #VP1.FCs.actual_revolutions;
NETWORK
TITLE = Sequence: Restart VP1 Protection
//only 12 times per hour
// >>test 30.0 sek, for production 300.0 sek
      L     3.000000e+02;
      T     #INTERNAL.RestartProtectTime;
//<<tests
//restart protection 
      A     #IF_FC_VP1.STATUS.STATE.Active;
      A     #VP1.motor_in_operation;
      FP    #INTERNAL.Flags.FP_VP1_ON.help;
      =     #TIMES.TOF_RestartProtectVP1.IN;
      CALL  "FC3 Timernachbildung" (
           in_Freigabe              := #TIMES.TOF_RestartProtectVP1.IN,
           in_Reset                 := FALSE,
           in_Impuls                := "M1.7 ClockTimerFunction",
           in_Impulszeit_in_100ms   := "MW 6 Timer Val Cycle FCs",
           in_Verzoegerungsart      := B#16#41,
           in_Verzoegerungszeit     := #INTERNAL.RestartProtectTime,
           io_Ausgangssignal        := #TIMES.TOF_RestartProtectVP1.Q,
           io_Zeitzaehler           := #TIMES.TOF_RestartProtectVP1.ET);
      L     #TIMES.TOF_RestartProtectVP1.ET;
      T     #HMI.PV.RestartIntervalVP1;
      L     #TIMES.TOF_RestartProtectVP1.ET;
      T     #HMI.PV.RestartIntervalVP1;
NETWORK
TITLE = Sequence: statuses to consumer
      A     #SEQUENCES.Sequence.AUTO;
      A     #IF_Consumer.CONTROL.CMD.Release;
      A     #VP1.motor_in_operation;
      A     #IF_FC_VP1.STATUS.STATE.Active;
      A     #FAValve.valve_in_operation;
      =     #SEQUENCES.Sequence.ACTIVE;
      A     #SEQUENCES.Sequence.ACTIVE;
      A     #IF_Consumer.STATUS.STATE.Ready;
      A     #IF_Consumer.CONTROL.CMD.Release;
      =     #IF_Consumer.STATUS.STATE.Active;
//pressure fault
//emty pressure reached
//actual pressure 
      L     #PressureVP1.PVAct;
//  L     -5.100000e+002
      T     #IF_Consumer.STATUS.ActualPressure;
      O     #VP1.fault;
      O     #IF_FC_VP1.STATUS.STATE.Fault;
      O     #FAValve.fault;
      O     #PressureVP1.OVErr;
      =     #IF_Consumer.STATUS.STATE.Fault;
NETWORK
TITLE = Call fresh air Valve
      CALL  "FC21 Ventil 1A0-2E" (
           in_Ventil_Typ            := 1,
           in_Handbedienung_erlaubt := TRUE,
           in_Quitt_Stoerung_noetig := FALSE,
           in_Quitt_Stoerung        := TRUE,
           in_Anlage_ein            := #i_xSystemActive,
           in_Ansteuerung_Ventil    := #FAValve.auto_mode_control,
           in_Eingang_angesteuert   := #i_xFAValveClose,
           in_Eingang_nicht_angest  := #i_xFAValveOpen,
           io_Ausgang_Ventil        := #q_xFAValve,
           io_Ventil_in_Betrieb     := #FAValve.valve_in_operation,
           io_Stoerung              := #f_xFAValve,
           io_Ventilstruktur        := #FAValve);	// service mode available from plc /  ack needed
      A     #FAValve.man_mode_control;
      =     #FAValve.man_mode_control;
NETWORK
TITLE = -------------------STATUS TO HMI--------------------------------
NETWORK
TITLE = Sequence: Restart block to HMI
      A     #TIMES.TOF_RestartProtectVP1.Q;
      AN    #VP1.motor_in_operation;
      =     #HMI.STATE.VP1Locked;
NETWORK
TITLE = ---- Interface ----
NETWORK
TITLE = interface FC
      CALL  "FC40 copy Obj-SST Master" (
           i_Freigabe               := #IF_FC_VP1.CONTROL.CMD.Request,
           i_Ziel_DB                := #IF_VP1_FC_DB,
           i_Ziel_DW                := #IF_VP1_FC_DW,
           i_SST_von_Ziel           := #IF_FC_VP1.STATUS,
           i_SST_an_Ziel            := #IF_FC_VP1.CONTROL,
           Ziel_frei                := #INTERNAL.IF.VP_FC.free);
NETWORK
TITLE = interface Consumer
      CALL  "FC41 copy Obj-SST Slave" (
           i_SST_von_Ziel           := #IF_Consumer.CONTROL,
           i_SST_an_Ziel            := #IF_Consumer.STATUS);
END_FUNCTION_BLOCK

FUNCTION_BLOCK "*** FCs ***"	// FB 4900
TITLE = Call Frequency Converters
//Creation:
//Date:            Author:                                               Version
//--------------------------------------------------------------------------------
//29.03.2018        ilia                                                 01.00.00
//
//Changes:
//No. Date:        Who       Description                           Mark   Version 
//--------------------------------------------------------------------------------
//01
//________________________________________________________________________________
//Function:
AUTHOR : ilia
NAME : project
VERSION : 1.0
BEGIN
NETWORK
TITLE = Vacuum Pump VP01
      CALL  "FREQ.CONVERTER" , "FC VACUUM PUMP" (
           in_FU_Typ                := 6,
           in_PEA_Adresse           := 1000,
           in_FU_Nummer             := 1,
           in_Motornennfrequenz     := 5.000000e+01,
           in_Motornenndrehzahl     := 1.455000e+03,
           aFU                      := "DB35 Acknolegments".Quittierung[200, 0],
           FU_Stoerung              := DB34.DBX 200.0);	//1.455000e+003
END_FUNCTION_BLOCK

FUNCTION_BLOCK "FREQ.CONVERTER"	// FB 4901
TITLE = FU Auswahlbaustein
//Erstellung:
//Datum        Bearbeiter                                                 Version
//--------------------------------------------------------------------------------
//10.07.06     Dominik Ilzhöfer (id)                                      01.00.00
//
//Änderungen:
//Nr. Datum    Bearb Änderung                                       Marke  Version
//--------------------------------------------------------------------------------
//01  06.11.07 sra   Motornennfrequenz und Motornenndrehzahl eingef.(001) 01.01.00
//02  23.07.13 sra   Status FU eingefügt                            (002) 01.02.00
//
//Baustein zur Ansteuerung von Frequenzumformern über Profibus-DB
//
//Parametrierung:
//FU-Typ:        wird zur richtigen Fehleranzeige an der Visualisierung benötigt
//               1=Siemens-MM4
//               2=SEW UFP11A
//               3=Lenze E82ZAFPC
//               4=Danfoss VLT5000
//               5=Danfoss FC300
//               6=SEW DFP21B
//             
//PEA-Adresse:   Anfangsadresse der Profibus-Schnittstelle
//Motordaten-DB: DB-Nummer mit Motordaten (Standard = DB4)
//FU-Nummer    : wird nur bei SEW Frequenzumformern mit UFP11A und DFP21B benötigt
//
//!Achtung!
//Bei den SEW Frequenzumformern wird die Motornennfrequenz und die 
//Motornenndrehzahl benötigt. D.h. es muss entweder ein Motordatensatz in dem 
//Motordaten-DB vorhanden sein oder die Werte müssen dem Baustein übergeben 
//werden.
NAME : standard
VERSION : 1.2
VAR_INPUT
  in_FU_Typ : INT ;	//1=Siemens-MM4, 2=SEW UFP11A, 3=Lenze E82ZAFPC, 4=Danfoss VLT5000
  in_PEA_Adresse : INT ;	//Basisadresse für EA-Daten im PEA-Bereich
  in_Motordaten_DB : INT  := 1;	//Adresse des DBs für Motordaten ( 0 = keine Motordaten schreiben )
  in_FU_Nummer : INT ;	//Nummer des FUs (für SEW-FUs)
  in_Motornennfrequenz : REAL ;	//muss bei SEW-FUs angegeben werden wenn kein Motordatensatz vorhanden ist
  in_Motornenndrehzahl : REAL ;	//muss bei SEW-FUs angegeben werden wenn kein Motordatensatz vorhanden ist
  aFU : BOOL ;
END_VAR
VAR_IN_OUT
  FU_Stoerung : BOOL ;
END_VAR
VAR
  reserve : ARRAY  [20 .. 29 ] OF BYTE ;
  Daten_Visualisierung : STRUCT
   von : STRUCT
    Quittierung_Stoerung : BOOL ;
    reserve : ARRAY  [2 .. 19 ] OF BYTE ;
   END_STRUCT ;
   an : STRUCT
    FU_Typ : INT ;
    Freigabe : BOOL ;
    Laeuft : BOOL ;
    Stoerung : BOOL ;
    Warnung : BOOL ;
    Sollfrequenz_erreicht : BOOL ;
    Sollfrequenz : REAL ;
    Istfrequenz : REAL ;
    Istdrehzahl : REAL ;
    Ausgangsstrom : REAL ;
    Leistung : REAL ;
    Drehmoment : REAL ;
    Spannung : REAL ;
    FU_Nummer : INT ;
    FB_Fehlermeldung : INT ;
    Stoerungsnummer : DINT ;
    reserve : ARRAY  [40 .. 47 ] OF BYTE ;
    Status : INT ;
   END_STRUCT ;
  END_STRUCT ;
  Schnittstelle : STRUCT
   von : STRUCT
    Antwort_DB : INT ;
    Antwort_DW : INT ;
    Sollfrequenz : REAL ;
    Motordatensatz_Nummer : INT ;
    reserve : ARRAY  [10 .. 17 ] OF BYTE ;
    Steuerbits : STRUCT
     Anforderung : BOOL ;
     Freigabe : BOOL ;
     Linkslauf : BOOL ;
    END_STRUCT ;
   END_STRUCT ;
   an : STRUCT
    Istfrequenz : REAL ;
    reserve : ARRAY  [4 .. 17 ] OF BYTE ;
    Statusbits : STRUCT
     Bereit : BOOL ;
     Laeuft : BOOL ;
     Stoerung : BOOL ;
    END_STRUCT ;
   END_STRUCT ;
  END_STRUCT ;
  Motordaten : STRUCT
   Nennleistugsfaktor : REAL ;
   Nennfrequenz : REAL ;
   Nenndrehzahl : REAL ;
   Nennstrom : REAL ;
   Nennspannung : REAL ;
   Nennleistung : REAL ;
   reserve : ARRAY  [24 .. 29 ] OF BYTE ;
  END_STRUCT ;
  Profibus_FB : FB 6119;
END_VAR
VAR_TEMP
  Motordaten_schreiben : BOOL ;
  Motordaten_Transfer_Fehl : INT ;
  Motordaten_Adresse_Quell : INT ;
  Motordaten_Adresse_Ziel : INT ;
END_VAR
BEGIN
NETWORK
TITLE = "Motordaten_schreiben" bilden
//Motordaten werden nur geschrieben, wenn ein Motordaten_DB und eine 
//Motordatensatz_Nummer ungleich 0 angegeben werden
      A(;
      L     #in_Motordaten_DB;
      L     0;
      <>I;
      );
      A(;
      L     #Schnittstelle.von.Motordatensatz_Nummer;
      L     0;
      <>I;
      );
      =     #Motordaten_schreiben;
NETWORK
TITLE = Motordatensatz in Motordaten kopieren
//Kompletter Motordatensatz wird aus Motordaten_DB kopiert
      L     #in_Motornennfrequenz;	// (001)
      T     #Motordaten.Nennfrequenz;	// (001)
      L     #in_Motornenndrehzahl;	// (001)
      T     #Motordaten.Nenndrehzahl;	// (001)
      A     #Motordaten_schreiben;
      JCN   SPR1;
      L     #Schnittstelle.von.Motordatensatz_Nummer;	// Nummer des Datensatzes des Motors
      L     -1;
      +I;
      L     30;	// Länge eines Datensatzes
      *I;
      T     #Motordaten_Adresse_Quell;	// Anfangsadresse des Datensatzes
      L     P##Motordaten;
      SRD   3;
      T     #Motordaten_Adresse_Ziel;
      CALL  "FC5 Blocktransfer" (
           Quell_Typ                := B#16#44,
           Quell_DB                 := #in_Motordaten_DB,
           Quell_DW                 := #Motordaten_Adresse_Quell,
           Ziel_Typ                 := B#16#49,
           Ziel_DB                  := 0,
           Ziel_DW                  := #Motordaten_Adresse_Ziel,
           Block_Laenge             := 24,
           outFehler                := #Motordaten_Transfer_Fehl);	// DB mit den Motordatensätzen /  Anfangsadresse des Datensatzes /  nicht verwendet da Ziel_Typ :='I' /  Abhängig vom Motordaten_DB
SPR1: NOP   0;
NETWORK
TITLE = Bei Anforderung "Bereit" bilden
      A     #Schnittstelle.von.Steuerbits.Anforderung;
      =     #Schnittstelle.an.Statusbits.Bereit;
NETWORK
TITLE = Auswahl des FU-Typs
//In der Multiinstanz "Profibus_FB" benötigten FU_Baustein im Datentyp angeben
      CALL  #Profibus_FB (
           in_PEA_Adresse           := #in_PEA_Adresse,
           in_FU_Nummer             := #in_FU_Nummer,
           in_Motordaten_J_N        := #Motordaten_schreiben,
           in_Freigabe              := #Schnittstelle.von.Steuerbits.Freigabe,
           in_Linkslauf             := #Schnittstelle.von.Steuerbits.Linkslauf,
           in_Quittierung_Stoerung  := #Daten_Visualisierung.von.Quittierung_Stoerung,
           in_Sollfrequenz          := #Schnittstelle.von.Sollfrequenz,
           in_Motorleistungsfaktor  := #Motordaten.Nennleistugsfaktor,
           in_Motornennfrequenz     := #Motordaten.Nennfrequenz,
           in_Motornenndrehzahl     := #Motordaten.Nenndrehzahl,
           in_Motornennstrom        := #Motordaten.Nennstrom,
           in_Motornennspannung     := #Motordaten.Nennspannung,
           in_Motornennleistung     := #Motordaten.Nennleistung,
           out_Istfrequenz          := #Daten_Visualisierung.an.Istfrequenz,
           out_Istdrehzahl          := #Daten_Visualisierung.an.Istdrehzahl,
           out_Leistung             := #Daten_Visualisierung.an.Leistung,
           out_Drehmoment           := #Daten_Visualisierung.an.Drehmoment,
           out_Motorspannung        := #Daten_Visualisierung.an.Spannung,
           out_Ausgangsstrom        := #Daten_Visualisierung.an.Ausgangsstrom,
           out_Stoerung             := #Daten_Visualisierung.an.Stoerung,
           out_Warnung              := #Daten_Visualisierung.an.Warnung,
           out_Sollwert_erreicht    := #Daten_Visualisierung.an.Sollfrequenz_erreicht,
           out_laeuft               := #Daten_Visualisierung.an.Laeuft,
           out_FB_Fehlermeldung     := #Daten_Visualisierung.an.FB_Fehlermeldung,
           out_Stoerungsnummer      := #Daten_Visualisierung.an.Stoerungsnummer);
NETWORK
TITLE = Verknüpfungen von Signalen für Visu und Schnittstelle
      L     #in_FU_Typ;
      T     #Daten_Visualisierung.an.FU_Typ;
      L     #in_FU_Nummer;
      T     #Daten_Visualisierung.an.FU_Nummer;
      A     #Schnittstelle.von.Steuerbits.Freigabe;
      =     #Daten_Visualisierung.an.Freigabe;
      L     #Schnittstelle.von.Sollfrequenz;
      T     #Daten_Visualisierung.an.Sollfrequenz;
      L     #Daten_Visualisierung.an.Istfrequenz;
      T     #Schnittstelle.an.Istfrequenz;
      A     #Daten_Visualisierung.an.Laeuft;
      =     #Schnittstelle.an.Statusbits.Laeuft;
      A     #Daten_Visualisierung.an.Stoerung;
      =     #Schnittstelle.an.Statusbits.Stoerung;
      =     #FU_Stoerung;
NETWORK
TITLE = Sollfrequenz löschen
      A     #Schnittstelle.von.Steuerbits.Freigabe;
      JC    M001;
      L     0;
      T     #Schnittstelle.von.Sollfrequenz;
      CLR;
      =     #Daten_Visualisierung.an.Sollfrequenz_erreicht;
M001: NOP   0;
NETWORK
TITLE = Statusanzeige für Visualisierung
//(002)
      L     16;	// Status Störung
      A     #Daten_Visualisierung.an.Stoerung;
      JC    Stat;
      L     13;	// Status Warnung
      A     #Daten_Visualisierung.an.Warnung;
      JC    Stat;
      L     5;	// Status läuft
      A     #Daten_Visualisierung.an.Laeuft;
      JC    Stat;
      L     1;	// Status aus
Stat: T     #Daten_Visualisierung.an.Status;
NETWORK
TITLE = Acknowledge FU Fault from the Visualization 
      A     #aFU;
      =     #Daten_Visualisierung.von.Quittierung_Stoerung;
NETWORK
TITLE = Schnittstellendaten kopieren
      CALL  "FC41 copy Obj-SST Slave" (
           i_SST_von_Ziel           := #Schnittstelle.von,
           i_SST_an_Ziel            := #Schnittstelle.an);
END_FUNCTION_BLOCK

